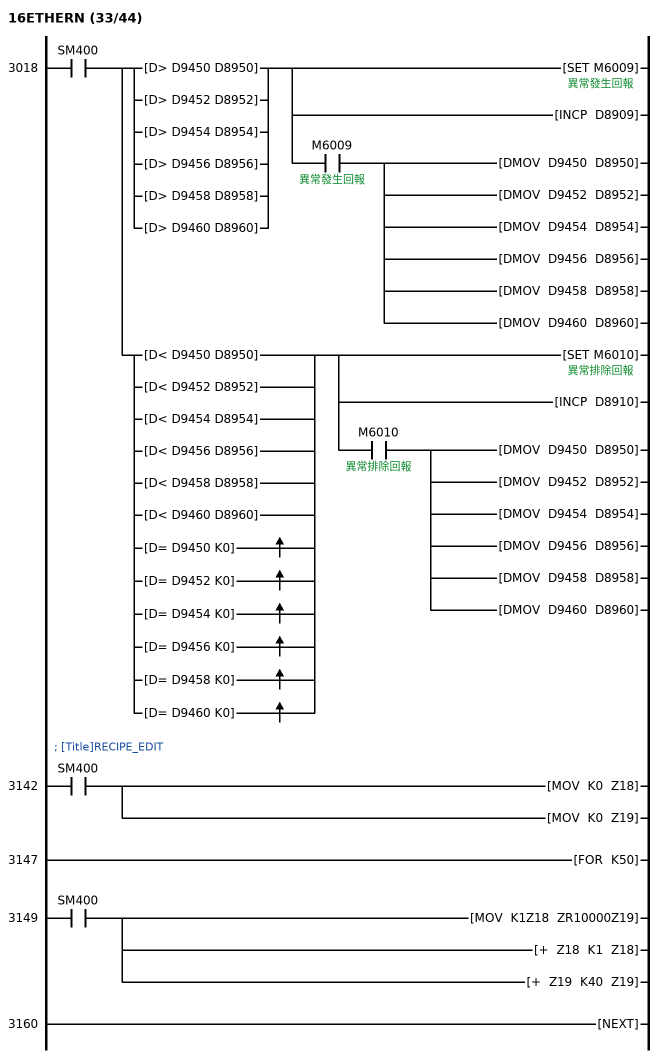
[picture p120: ladder of 16ETHERN, rungs at steps 3018 to 3160]
3018  LD      SM400
      MPS
      LDD>    D9450 D8950
      ORD>    D9452 D8952
      ORD>    D9454 D8954
      ORD>    D9456 D8956
      ORD>    D9458 D8958
      ORD>    D9460 D8960
      ANB
      SET     M6009  ; 異常發生回報
      INCP    D8909
      AND     M6009  ; 異常發生回報
      DMOV    D9450 D8950
      DMOV    D9452 D8952
      DMOV    D9454 D8954
      DMOV    D9456 D8956
      DMOV    D9458 D8958
      DMOV    D9460 D8960
      MPP
      LDD<    D9450 D8950
      ORD<    D9452 D8952
      ORD<    D9454 D8954
      ORD<    D9456 D8956
      ORD<    D9458 D8958
      ORD<    D9460 D8960
      LDD=    D9450 K0
      MEP
      ORB
      LDD=    D9452 K0
      MEP
      ORB
      LDD=    D9454 K0
      MEP
      ORB
      LDD=    D9456 K0
      MEP
      ORB
      LDD=    D9458 K0
      MEP
      ORB
      LDD=    D9460 K0
      MEP
      ORB
      ANB
      SET     M6010  ; 異常排除回報
      INCP    D8910
      AND     M6010  ; 異常排除回報
      DMOV    D9450 D8950
      DMOV    D9452 D8952
      DMOV    D9454 D8954
      DMOV    D9456 D8956
      DMOV    D9458 D8958
      DMOV    D9460 D8960
; [Title]RECIPE_EDIT
3142  LD      SM400
      MOV     K0 Z18
      MOV     K0 Z19
3147  FOR     K50
3149  LD      SM400
      MOV     K1Z18 ZR10000Z19
      +       Z18 K1 Z18
      +       Z19 K40 Z19
3160  NEXT
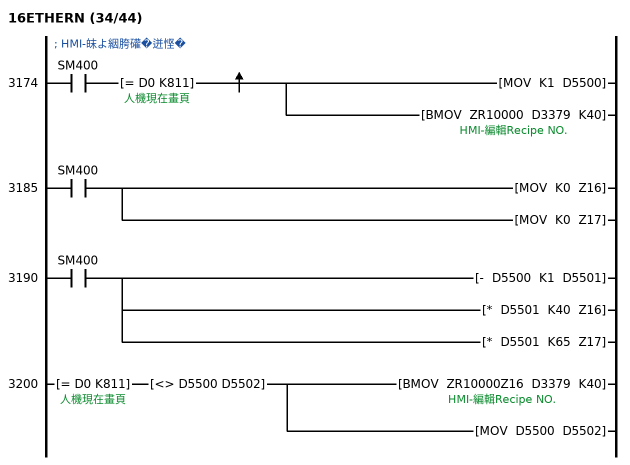
; HMI-配方編輯畫面顯示
3174  LD      SM400
      AND=    D0 K811  ; 人機現在畫頁
      MEP
      MOV     K1 D5500
      BMOV    ZR10000 D3379 K40  ; HMI-編輯Recipe NO.
3185  LD      SM400
      MOV     K0 Z16
      MOV     K0 Z17
3190  LD      SM400
      -       D5500 K1 D5501
      *       D5501 K40 Z16
      *       D5501 K65 Z17
3200  LD=     D0 K811  ; 人機現在畫頁
      AND<>   D5500 D5502
      BMOV    ZR10000Z16 D3379 K40
      MOV     D5500 D5502
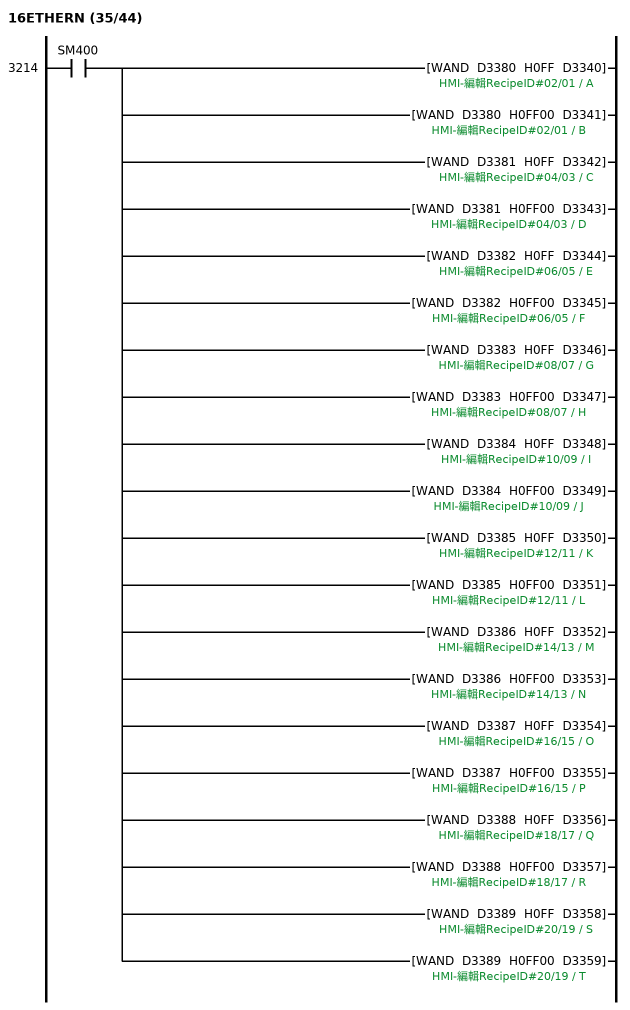
3214  LD      SM400
      WAND    D3380 H0FF D3340  ; HMI-編輯RecipeID#02/01 / A
      WAND    D3380 H0FF00 D3341  ; B
      WAND    D3381 H0FF D3342  ; HMI-編輯RecipeID#04/03 / C
      WAND    D3381 H0FF00 D3343  ; D
      WAND    D3382 H0FF D3344  ; HMI-編輯RecipeID#06/05 / E
      WAND    D3382 H0FF00 D3345  ; F
      WAND    D3383 H0FF D3346  ; HMI-編輯RecipeID#08/07 / G
      WAND    D3383 H0FF00 D3347  ; H
      WAND    D3384 H0FF D3348  ; HMI-編輯RecipeID#10/09 / I
      WAND    D3384 H0FF00 D3349  ; J
      WAND    D3385 H0FF D3350  ; HMI-編輯RecipeID#12/11 / K
      WAND    D3385 H0FF00 D3351  ; L
      WAND    D3386 H0FF D3352  ; HMI-編輯RecipeID#14/13 / M
      WAND    D3386 H0FF00 D3353  ; N
      WAND    D3387 H0FF D3354  ; HMI-編輯RecipeID#16/15 / O
      WAND    D3387 H0FF00 D3355  ; P
      WAND    D3388 H0FF D3356  ; HMI-編輯RecipeID#18/17 / Q
      WAND    D3388 H0FF00 D3357  ; R
      WAND    D3389 H0FF D3358  ; HMI-編輯RecipeID#20/19 / S
      WAND    D3389 H0FF00 D3359  ; T
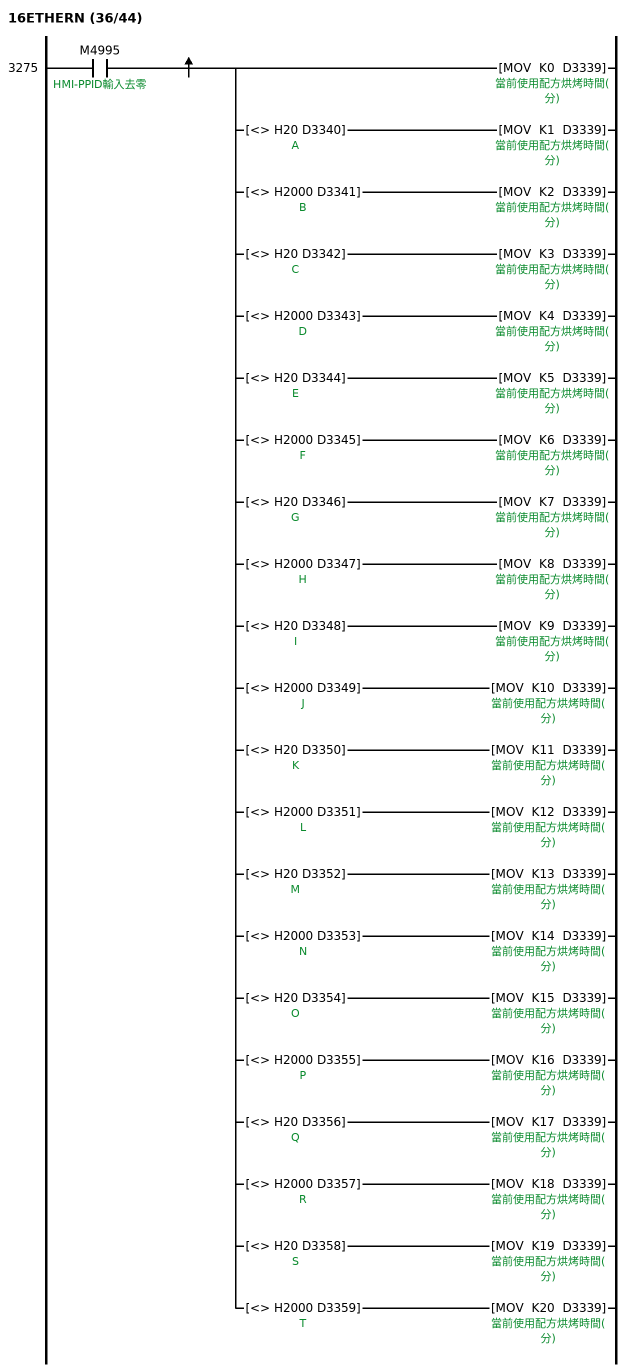
3275  LD      M4995  ; HMI-PPID輸入去零
      MEP
      MOV     K0 D3339  ; 當前使用配方烘烤時間(分)
      MPS
      AND<>   H20 D3340  ; A
      MOV     K1 D3339
      MRD
      AND<>   H2000 D3341  ; B
      MOV     K2 D3339
      MRD
      AND<>   H20 D3342  ; C
      MOV     K3 D3339
      MRD
      AND<>   H2000 D3343  ; D
      MOV     K4 D3339
      MRD
      AND<>   H20 D3344  ; E
      MOV     K5 D3339
      MRD
      AND<>   H2000 D3345  ; F
      MOV     K6 D3339
      MRD
      AND<>   H20 D3346  ; G
      MOV     K7 D3339
      MRD
      AND<>   H2000 D3347  ; H
      MOV     K8 D3339
      MRD
      AND<>   H20 D3348  ; I
      MOV     K9 D3339
      MRD
      AND<>   H2000 D3349  ; J
      MOV     K10 D3339
      MRD
      AND<>   H20 D3350  ; K
      MOV     K11 D3339
      MRD
      AND<>   H2000 D3351  ; L
      MOV     K12 D3339
      MRD
      AND<>   H20 D3352  ; M
      MOV     K13 D3339
      MRD
      AND<>   H2000 D3353  ; N
      MOV     K14 D3339
      MRD
      AND<>   H20 D3354  ; O
      MOV     K15 D3339
      MRD
      AND<>   H2000 D3355  ; P
      MOV     K16 D3339
      MRD
      AND<>   H20 D3356  ; Q
      MOV     K17 D3339
      MRD
      AND<>   H2000 D3357  ; R
      MOV     K18 D3339
      MRD
      AND<>   H20 D3358  ; S
      MOV     K19 D3339
      MPP
      AND<>   H2000 D3359  ; T
      MOV     K20 D3339
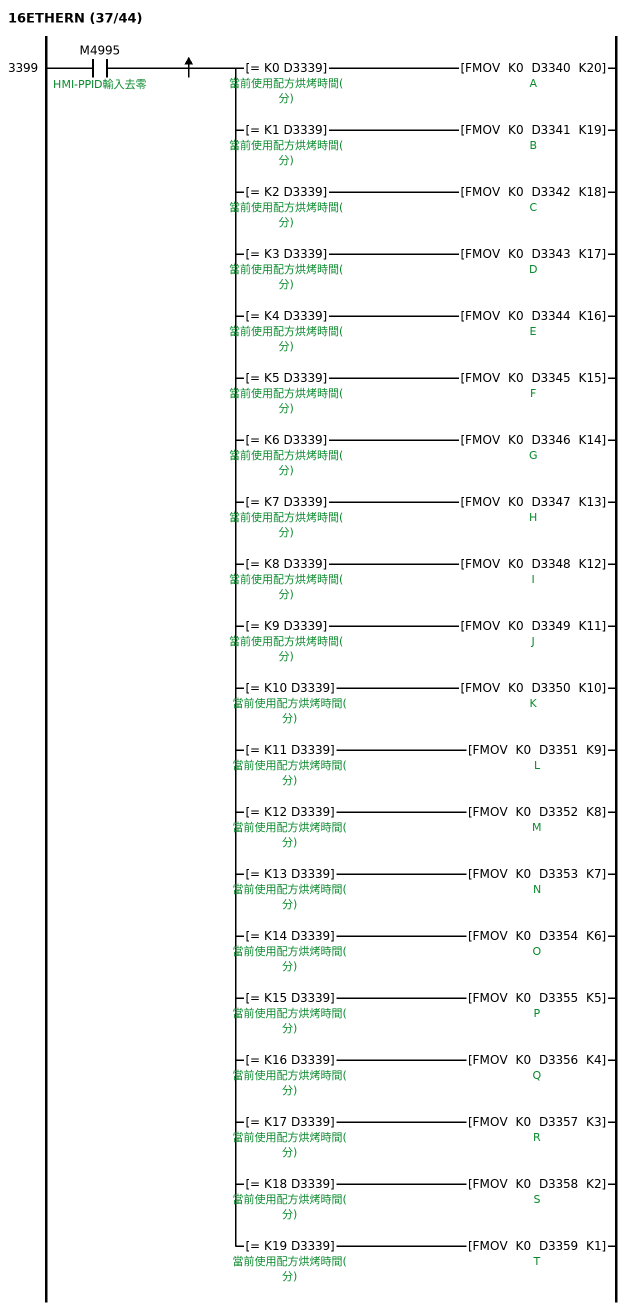
3399  LD      M4995  ; HMI-PPID輸入去零
      MEP
      MPS
      AND=    K0 D3339  ; 當前使用配方烘烤時間(分)
      FMOV    K0 D3340 K20
      MRD
      AND=    K1 D3339  ; 當前使用配方烘烤時間(分)
      FMOV    K0 D3341 K19
      MRD
      AND=    K2 D3339  ; 當前使用配方烘烤時間(分)
      FMOV    K0 D3342 K18
      MRD
      AND=    K3 D3339  ; 當前使用配方烘烤時間(分)
      FMOV    K0 D3343 K17
      MRD
      AND=    K4 D3339  ; 當前使用配方烘烤時間(分)
      FMOV    K0 D3344 K16
      MRD
      AND=    K5 D3339  ; 當前使用配方烘烤時間(分)
      FMOV    K0 D3345 K15
      MRD
      AND=    K6 D3339  ; 當前使用配方烘烤時間(分)
      FMOV    K0 D3346 K14
      MRD
      AND=    K7 D3339  ; 當前使用配方烘烤時間(分)
      FMOV    K0 D3347 K13
      MRD
      AND=    K8 D3339  ; 當前使用配方烘烤時間(分)
      FMOV    K0 D3348 K12
      MRD
      AND=    K9 D3339  ; 當前使用配方烘烤時間(分)
      FMOV    K0 D3349 K11
      MRD
      AND=    K10 D3339  ; 當前使用配方烘烤時間(分)
      FMOV    K0 D3350 K10
      MRD
      AND=    K11 D3339  ; 當前使用配方烘烤時間(分)
      FMOV    K0 D3351 K9
      MRD
      AND=    K12 D3339  ; 當前使用配方烘烤時間(分)
      FMOV    K0 D3352 K8
      MRD
      AND=    K13 D3339  ; 當前使用配方烘烤時間(分)
      FMOV    K0 D3353 K7
      MRD
      AND=    K14 D3339  ; 當前使用配方烘烤時間(分)
      FMOV    K0 D3354 K6
      MRD
      AND=    K15 D3339  ; 當前使用配方烘烤時間(分)
      FMOV    K0 D3355 K5
      MRD
      AND=    K16 D3339  ; 當前使用配方烘烤時間(分)
      FMOV    K0 D3356 K4
      MRD
      AND=    K17 D3339  ; 當前使用配方烘烤時間(分)
      FMOV    K0 D3357 K3
      MRD
      AND=    K18 D3339  ; 當前使用配方烘烤時間(分)
      FMOV    K0 D3358 K2
      MPP
      AND=    K19 D3339  ; 當前使用配方烘烤時間(分)
      FMOV    K0 D3359 K1
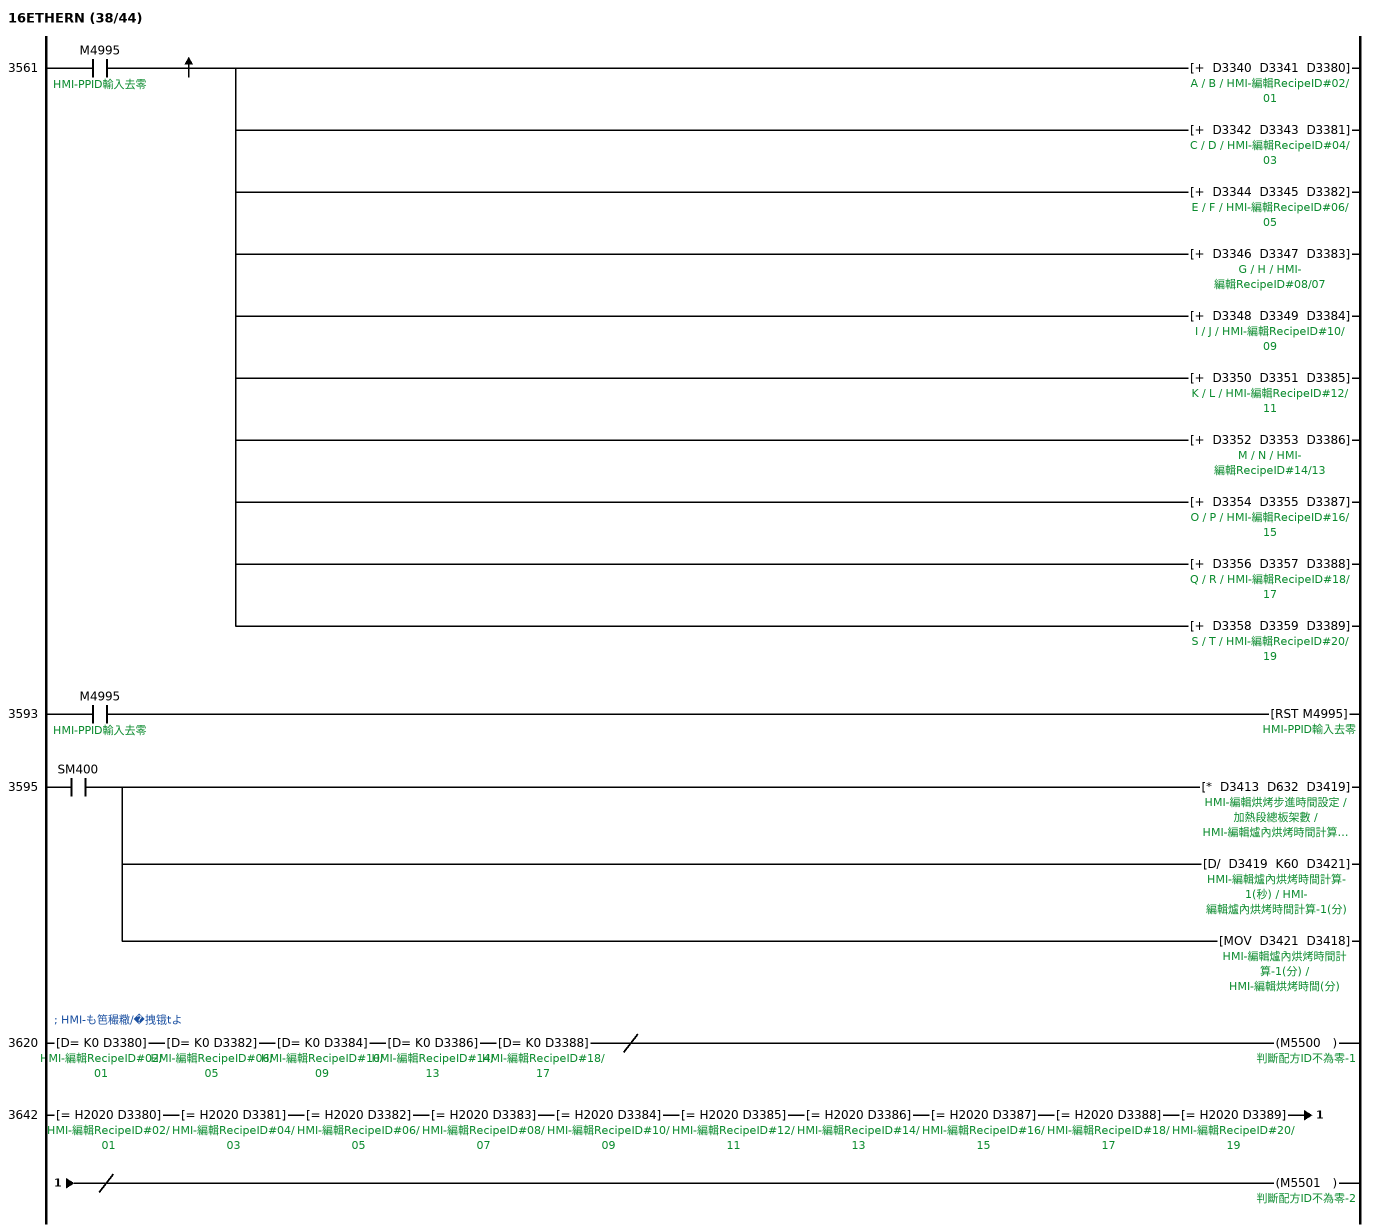
3561  LD      M4995  ; HMI-PPID輸入去零
      MEP
      +       D3340 D3341 D3380
      +       D3342 D3343 D3381
      +       D3344 D3345 D3382
      +       D3346 D3347 D3383
      +       D3348 D3349 D3384
      +       D3350 D3351 D3385
      +       D3352 D3353 D3386
      +       D3354 D3355 D3387
      +       D3356 D3357 D3388
      +       D3358 D3359 D3389
3593  LD      M4995  ; HMI-PPID輸入去零
      RST     M4995  ; HMI-PPID輸入去零
3595  LD      SM400
      *       D3413 D632 D3419  ; HMI-編輯烘烤步進時間設定 / 加熱段總板架數 / HMI-編輯爐內烘烤時間計算-1(秒)
      D/      D3419 K60 D3421  ; HMI-編輯爐內烘烤時間計算-1(分)
      MOV     D3421 D3418  ; HMI-編輯烘烤時間(分)
; HMI-手動新增/修改配方
3620  LDD=    K0 D3380  ; HMI-編輯RecipeID#02/01
      ANDD=   K0 D3382  ; HMI-編輯RecipeID#06/05
      ANDD=   K0 D3384  ; HMI-編輯RecipeID#10/09
      ANDD=   K0 D3386  ; HMI-編輯RecipeID#14/13
      ANDD=   K0 D3388  ; HMI-編輯RecipeID#18/17
      INV
      OUT     M5500  ; 判斷配方ID不為零-1
3642  LD=     H2020 D3380  ; HMI-編輯RecipeID#02/01
      AND=    H2020 D3381  ; HMI-編輯RecipeID#04/03
      AND=    H2020 D3382  ; HMI-編輯RecipeID#06/05
      AND=    H2020 D3383  ; HMI-編輯RecipeID#08/07
      AND=    H2020 D3384  ; HMI-編輯RecipeID#10/09
      AND=    H2020 D3385  ; HMI-編輯RecipeID#12/11
      AND=    H2020 D3386  ; HMI-編輯RecipeID#14/13
      AND=    H2020 D3387  ; HMI-編輯RecipeID#16/15
      AND=    H2020 D3388  ; HMI-編輯RecipeID#18/17
      AND=    H2020 D3389  ; HMI-編輯RecipeID#20/19
      INV
      OUT     M5501  ; 判斷配方ID不為零-2
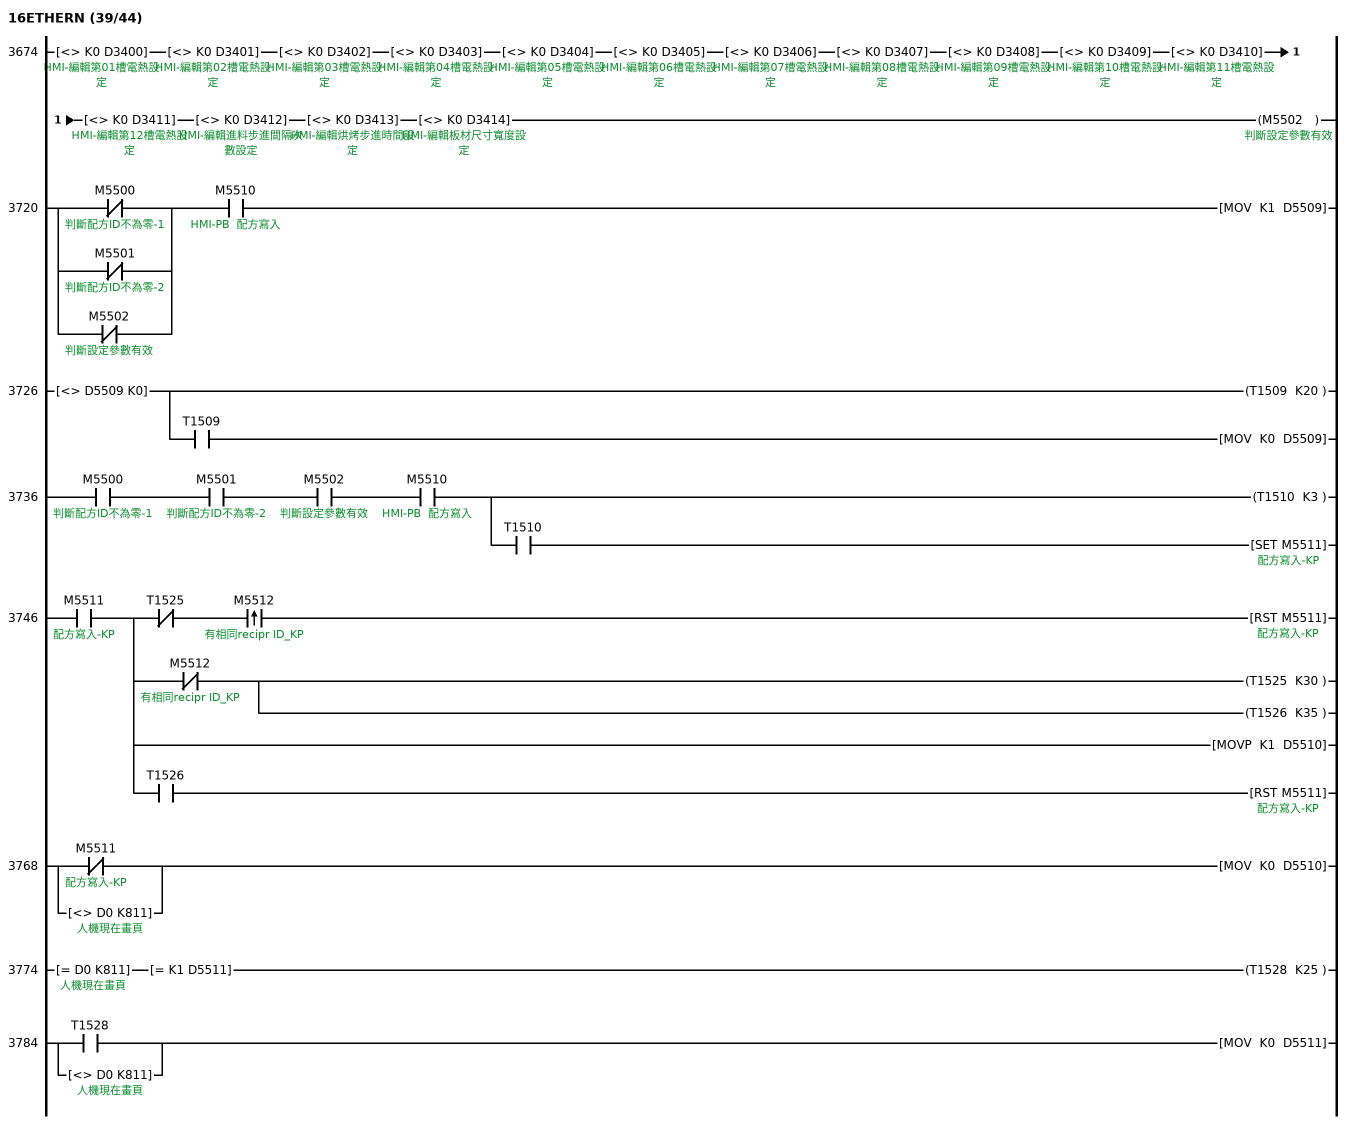
3674  LD<>    K0 D3400  ; HMI-編輯第01槽電熱設定
      AND<>   K0 D3401  ; HMI-編輯第02槽電熱設定
      AND<>   K0 D3402  ; HMI-編輯第03槽電熱設定
      AND<>   K0 D3403  ; HMI-編輯第04槽電熱設定
      AND<>   K0 D3404  ; HMI-編輯第05槽電熱設定
      AND<>   K0 D3405  ; HMI-編輯第06槽電熱設定
      AND<>   K0 D3406  ; HMI-編輯第07槽電熱設定
      AND<>   K0 D3407  ; HMI-編輯第08槽電熱設定
      AND<>   K0 D3408  ; HMI-編輯第09槽電熱設定
      AND<>   K0 D3409  ; HMI-編輯第10槽電熱設定
      AND<>   K0 D3410  ; HMI-編輯第11槽電熱設定
      AND<>   K0 D3411  ; HMI-編輯第12槽電熱設定
      AND<>   K0 D3412  ; HMI-編輯進料步進間隔次數設定
      AND<>   K0 D3413  ; HMI-編輯烘烤步進時間設定
      AND<>   K0 D3414  ; HMI-編輯板材尺寸寬度設定
      OUT     M5502  ; 判斷設定參數有效
3720  LDI     M5500  ; 判斷配方ID不為零-1
      ORI     M5501  ; 判斷配方ID不為零-2
      ORI     M5502  ; 判斷設定參數有效
      AND     M5510  ; HMI-PB  配方寫入
      MOV     K1 D5509
3726  LD<>    D5509 K0
      OUT     T1509 K20
      AND     T1509
      MOV     K0 D5509
3736  LD      M5500  ; 判斷配方ID不為零-1
      AND     M5501  ; 判斷配方ID不為零-2
      AND     M5502  ; 判斷設定參數有效
      AND     M5510  ; HMI-PB  配方寫入
      OUT     T1510 K3
      AND     T1510
      SET     M5511  ; 配方寫入-KP
3746  LD      M5511  ; 配方寫入-KP
      MPS
      ANI     T1525
      ANDP    M5512  ; 有相同recipr ID_KP
      RST     M5511  ; 配方寫入-KP
      MRD
      ANI     M5512  ; 有相同recipr ID_KP
      OUT     T1525 K30
      OUT     T1526 K35
      MPP
      MOVP    K1 D5510
      AND     T1526
      RST     M5511  ; 配方寫入-KP
3768  LDI     M5511  ; 配方寫入-KP
      OR<>    D0 K811  ; 人機現在畫頁
      MOV     K0 D5510
3774  LD=     D0 K811  ; 人機現在畫頁
      AND=    K1 D5511
      OUT     T1528 K25
3784  LD      T1528
      OR<>    D0 K811  ; 人機現在畫頁
      MOV     K0 D5511
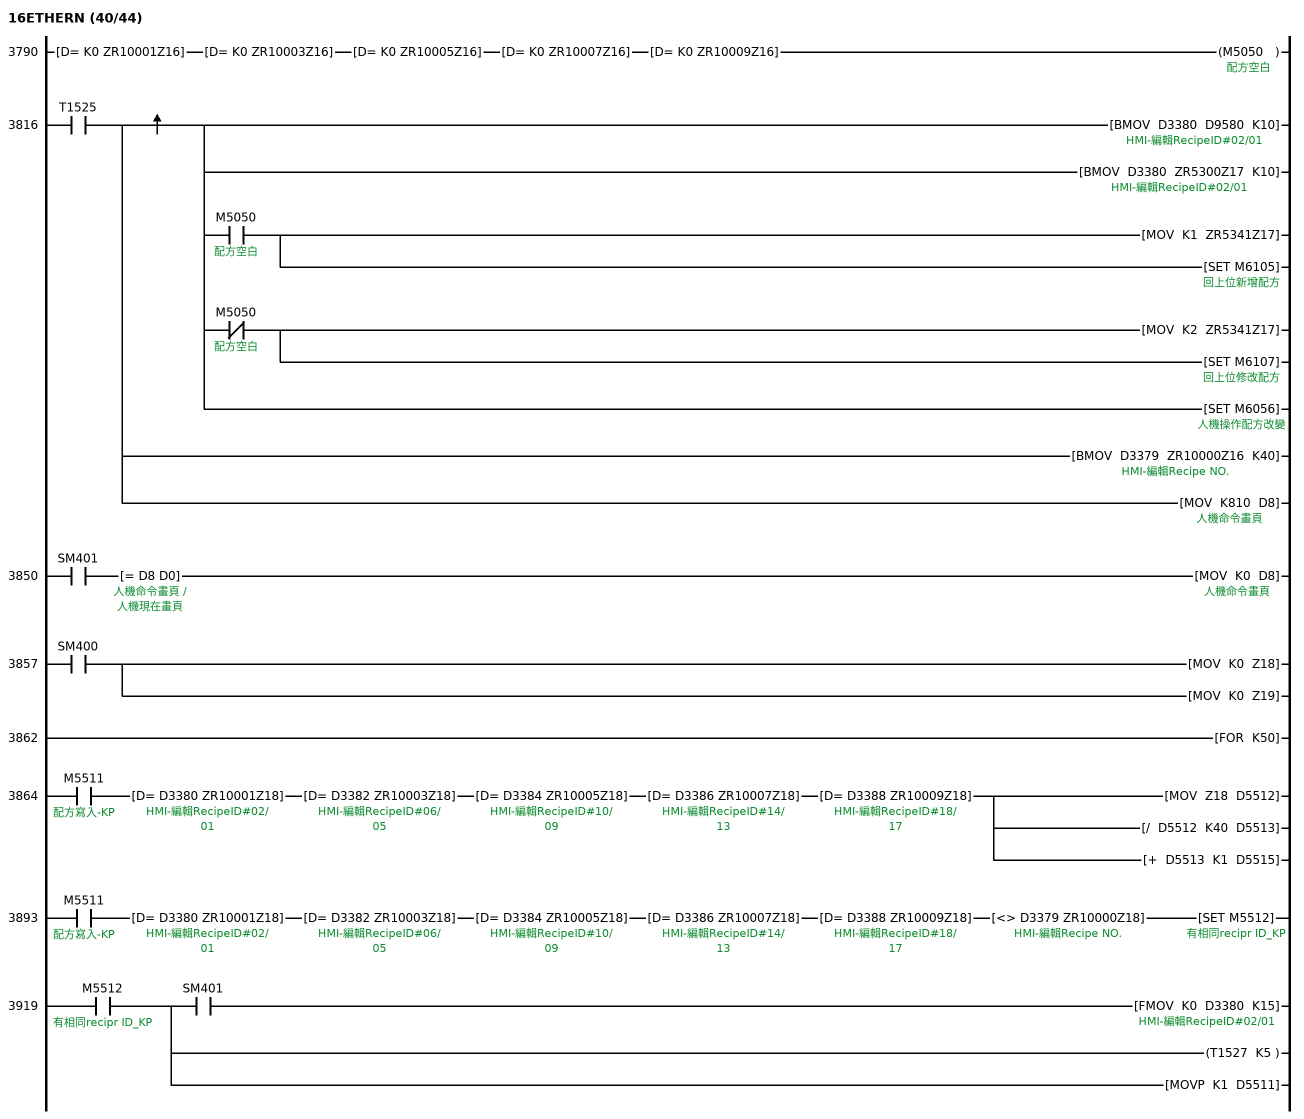
3790  LDD=    K0 ZR10001Z16
      ANDD=   K0 ZR10003Z16
      ANDD=   K0 ZR10005Z16
      ANDD=   K0 ZR10007Z16
      ANDD=   K0 ZR10009Z16
      OUT     M5050  ; 配方空白
3816  LD      T1525
      MPS
      MEP
      BMOV    D3380 D9580 K10
      BMOV    D3380 ZR5300Z17 K10
      MPS
      AND     M5050  ; 配方空白
      MOV     K1 ZR5341Z17
      SET     M6105  ; 回上位新增配方
      MRD
      ANI     M5050  ; 配方空白
      MOV     K2 ZR5341Z17
      SET     M6107  ; 回上位修改配方
      MPP
      SET     M6056  ; 人機操作配方改變
      MPP
      BMOV    D3379 ZR10000Z16 K40
      MOV     K810 D8
3850  LD      SM401
      AND=    D8 D0  ; 人機命令畫頁 / 人機現在畫頁
      MOV     K0 D8
3857  LD      SM400
      MOV     K0 Z18
      MOV     K0 Z19
3862  FOR     K50
3864  LD      M5511  ; 配方寫入-KP
      ANDD=   D3380 ZR10001Z18  ; HMI-編輯RecipeID#02/01
      ANDD=   D3382 ZR10003Z18  ; HMI-編輯RecipeID#06/05
      ANDD=   D3384 ZR10005Z18  ; HMI-編輯RecipeID#10/09
      ANDD=   D3386 ZR10007Z18  ; HMI-編輯RecipeID#14/13
      ANDD=   D3388 ZR10009Z18  ; HMI-編輯RecipeID#18/17
      MOV     Z18 D5512
      /       D5512 K40 D5513
      +       D5513 K1 D5515
3893  LD      M5511  ; 配方寫入-KP
      ANDD=   D3380 ZR10001Z18  ; HMI-編輯RecipeID#02/01
      ANDD=   D3382 ZR10003Z18  ; HMI-編輯RecipeID#06/05
      ANDD=   D3384 ZR10005Z18  ; HMI-編輯RecipeID#10/09
      ANDD=   D3386 ZR10007Z18  ; HMI-編輯RecipeID#14/13
      ANDD=   D3388 ZR10009Z18  ; HMI-編輯RecipeID#18/17
      AND<>   D3379 ZR10000Z18  ; HMI-編輯Recipe NO.
      SET     M5512  ; 有相同recipr ID_KP
3919  LD      M5512  ; 有相同recipr ID_KP
      MPS
      AND     SM401
      FMOV    K0 D3380 K15
      MPP
      OUT     T1527 K5
      MOVP    K1 D5511
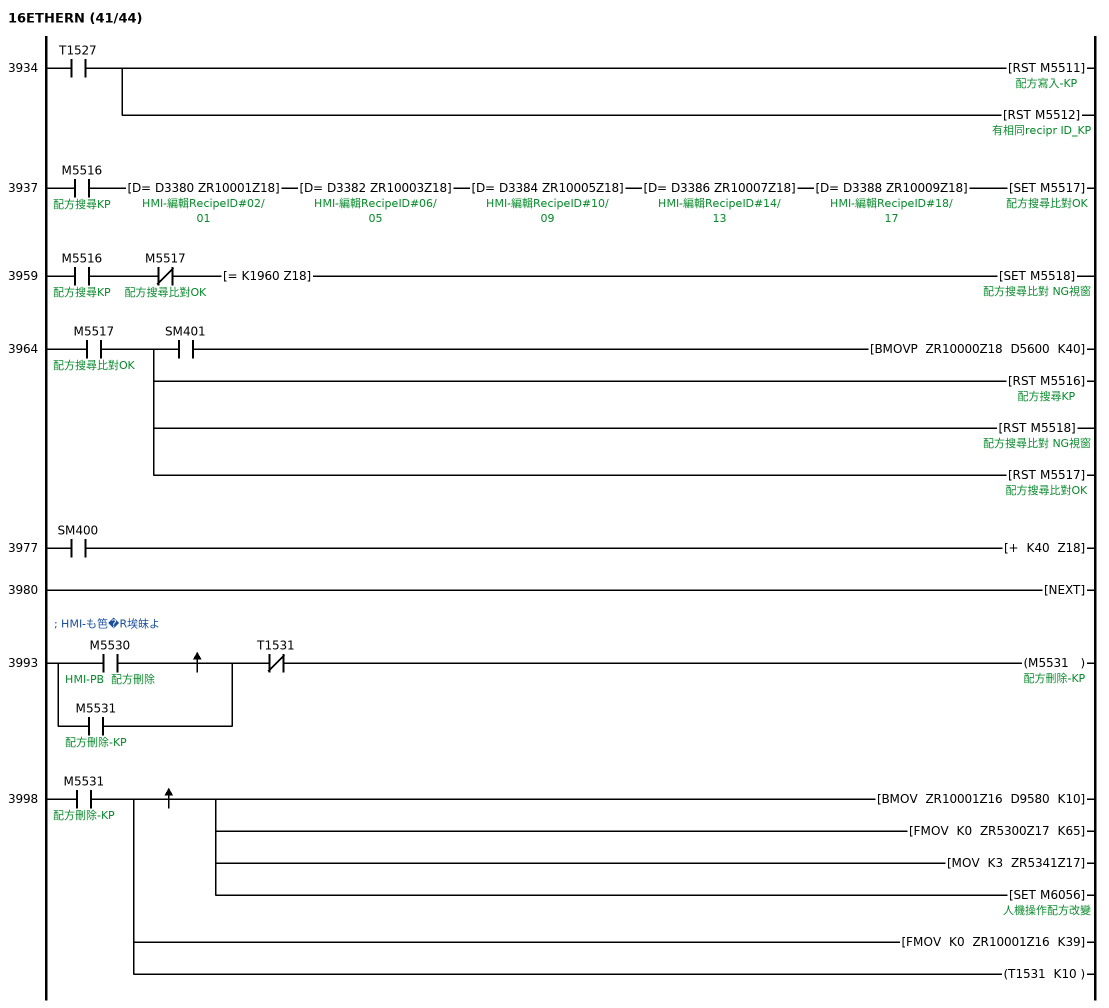
3934  LD      T1527
      RST     M5511  ; 配方寫入-KP
      RST     M5512  ; 有相同recipr ID_KP
3937  LD      M5516  ; 配方搜尋KP
      ANDD=   D3380 ZR10001Z18  ; HMI-編輯RecipeID#02/01
      ANDD=   D3382 ZR10003Z18  ; HMI-編輯RecipeID#06/05
      ANDD=   D3384 ZR10005Z18  ; HMI-編輯RecipeID#10/09
      ANDD=   D3386 ZR10007Z18  ; HMI-編輯RecipeID#14/13
      ANDD=   D3388 ZR10009Z18  ; HMI-編輯RecipeID#18/17
      SET     M5517  ; 配方搜尋比對OK
3959  LD      M5516  ; 配方搜尋KP
      ANI     M5517  ; 配方搜尋比對OK
      AND=    K1960 Z18
      SET     M5518  ; 配方搜尋比對 NG視窗
3964  LD      M5517  ; 配方搜尋比對OK
      MPS
      AND     SM401
      BMOVP   ZR10000Z18 D5600 K40
      MPP
      RST     M5516  ; 配方搜尋KP
      RST     M5518  ; 配方搜尋比對 NG視窗
      RST     M5517  ; 配方搜尋比對OK
3977  LD      SM400
      +       K40 Z18
3980  NEXT
; HMI-手動刪除配方
3993  LD      M5530  ; HMI-PB  配方刪除
      MEP
      OR      M5531  ; 配方刪除-KP
      ANI     T1531
      OUT     M5531  ; 配方刪除-KP
3998  LD      M5531  ; 配方刪除-KP
      MPS
      MEP
      BMOV    ZR10001Z16 D9580 K10
      FMOV    K0 ZR5300Z17 K65
      MOV     K3 ZR5341Z17
      SET     M6056  ; 人機操作配方改變
      MPP
      FMOV    K0 ZR10001Z16 K39
      OUT     T1531 K10
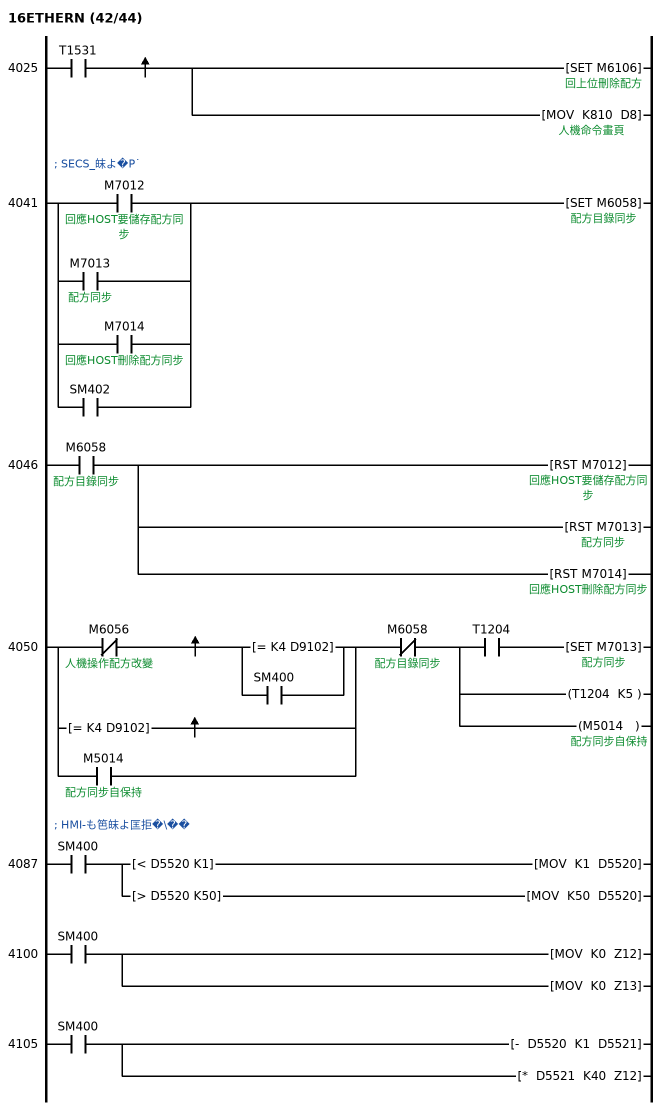
4025  LD      T1531
      MEP
      SET     M6106  ; 回上位刪除配方
      MOV     K810 D8
; SECS_配方同步
4041  LD      M7012  ; 回應HOST要儲存配方同步
      OR      M7013  ; 配方同步
      OR      M7014  ; 回應HOST刪除配方同步
      OR      SM402
      SET     M6058  ; 配方目錄同步
4046  LD      M6058  ; 配方目錄同步
      RST     M7012  ; 回應HOST要儲存配方同步
      RST     M7013  ; 配方同步
      RST     M7014  ; 回應HOST刪除配方同步
4050  LDI     M6056  ; 人機操作配方改變
      MEP
      LD=     K4 D9102
      OR      SM400
      ANB
      LD=     K4 D9102
      MEP
      ORB
      OR      M5014  ; 配方同步自保持
      ANI     M6058  ; 配方目錄同步
      MPS
      AND     T1204
      SET     M7013  ; 配方同步
      MPP
      OUT     T1204 K5
      OUT     M5014  ; 配方同步自保持
; HMI-手動配方選擇功能
4087  LD      SM400
      MPS
      AND<    D5520 K1
      MOV     K1 D5520
      MPP
      AND>    D5520 K50
      MOV     K50 D5520
4100  LD      SM400
      MOV     K0 Z12
      MOV     K0 Z13
4105  LD      SM400
      -       D5520 K1 D5521
      *       D5521 K40 Z12
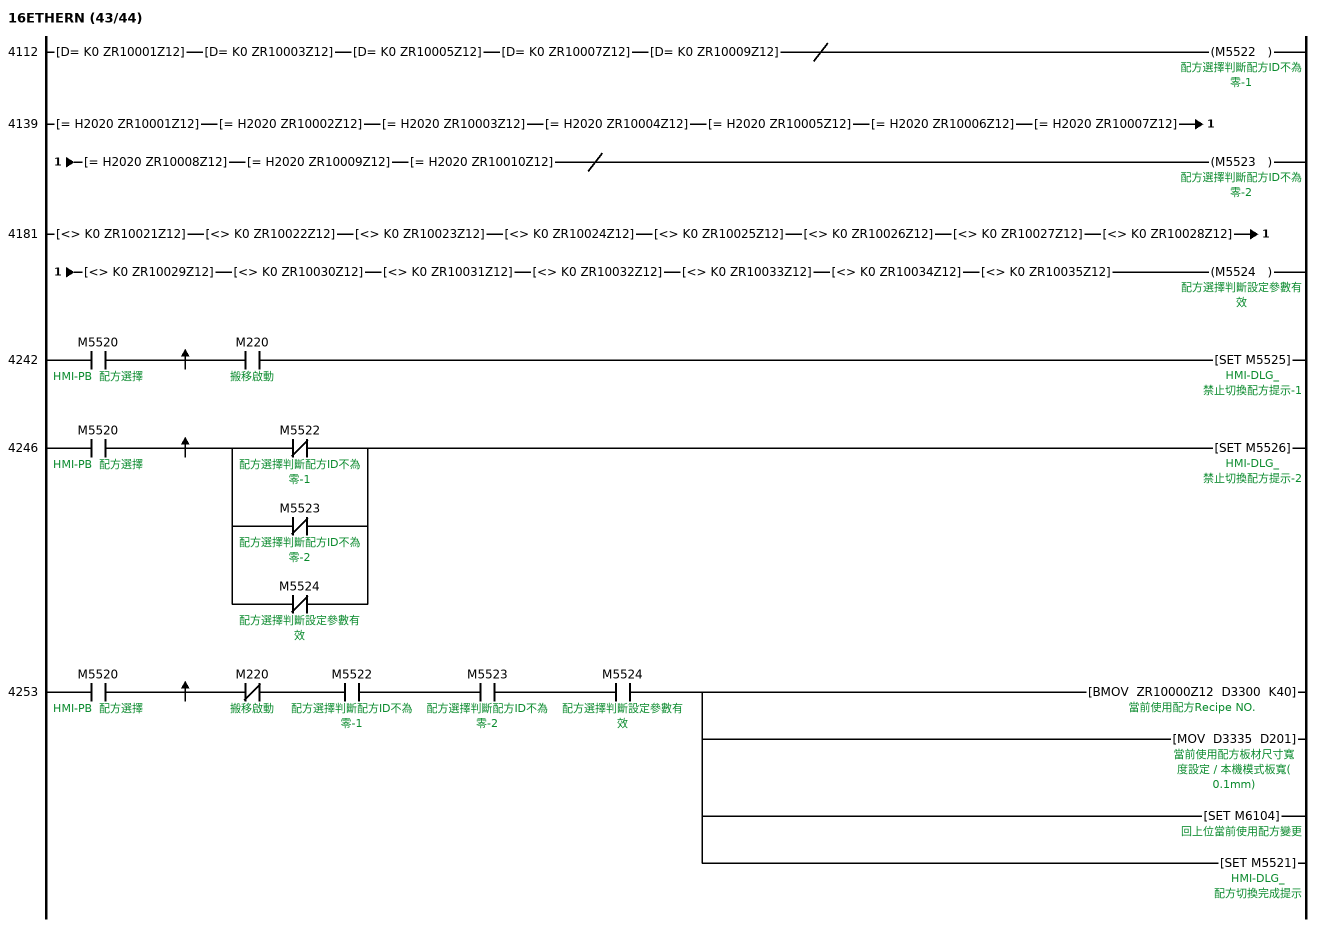
4112  LDD=    K0 ZR10001Z12
      ANDD=   K0 ZR10003Z12
      ANDD=   K0 ZR10005Z12
      ANDD=   K0 ZR10007Z12
      ANDD=   K0 ZR10009Z12
      INV
      OUT     M5522  ; 配方選擇判斷配方ID不為零-1
4139  LD=     H2020 ZR10001Z12
      AND=    H2020 ZR10002Z12
      AND=    H2020 ZR10003Z12
      AND=    H2020 ZR10004Z12
      AND=    H2020 ZR10005Z12
      AND=    H2020 ZR10006Z12
      AND=    H2020 ZR10007Z12
      AND=    H2020 ZR10008Z12
      AND=    H2020 ZR10009Z12
      AND=    H2020 ZR10010Z12
      INV
      OUT     M5523  ; 配方選擇判斷配方ID不為零-2
4181  LD<>    K0 ZR10021Z12
      AND<>   K0 ZR10022Z12
      AND<>   K0 ZR10023Z12
      AND<>   K0 ZR10024Z12
      AND<>   K0 ZR10025Z12
      AND<>   K0 ZR10026Z12
      AND<>   K0 ZR10027Z12
      AND<>   K0 ZR10028Z12
      AND<>   K0 ZR10029Z12
      AND<>   K0 ZR10030Z12
      AND<>   K0 ZR10031Z12
      AND<>   K0 ZR10032Z12
      AND<>   K0 ZR10033Z12
      AND<>   K0 ZR10034Z12
      AND<>   K0 ZR10035Z12
      OUT     M5524  ; 配方選擇判斷設定參數有效
4242  LD      M5520  ; HMI-PB  配方選擇
      MEP
      AND     M220  ; 搬移啟動
      SET     M5525  ; HMI-DLG_禁止切換配方提示-1
4246  LD      M5520  ; HMI-PB  配方選擇
      MEP
      LDI     M5522  ; 配方選擇判斷配方ID不為零-1
      ORI     M5523  ; 配方選擇判斷配方ID不為零-2
      ORI     M5524  ; 配方選擇判斷設定參數有效
      ANB
      SET     M5526  ; HMI-DLG_禁止切換配方提示-2
4253  LD      M5520  ; HMI-PB  配方選擇
      MEP
      ANI     M220  ; 搬移啟動
      AND     M5522  ; 配方選擇判斷配方ID不為零-1
      AND     M5523  ; 配方選擇判斷配方ID不為零-2
      AND     M5524  ; 配方選擇判斷設定參數有效
      BMOV    ZR10000Z12 D3300 K40
      MOV     D3335 D201
      SET     M6104  ; 回上位當前使用配方變更
      SET     M5521  ; HMI-DLG_配方切換完成提示
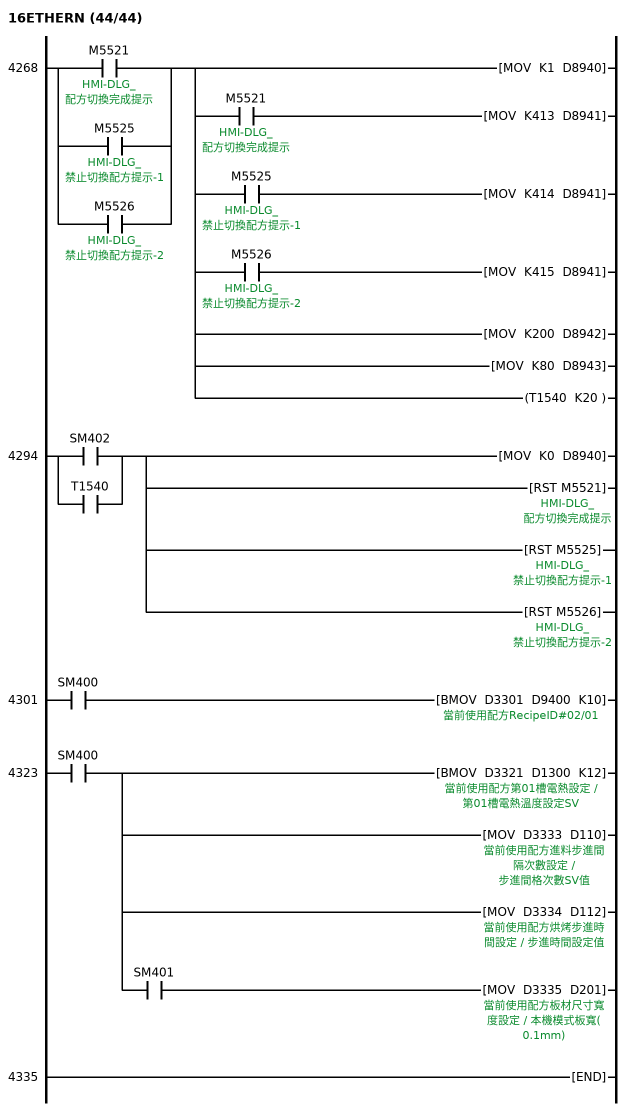
4268  LD      M5521  ; HMI-DLG_配方切換完成提示
      OR      M5525  ; HMI-DLG_禁止切換配方提示-1
      OR      M5526  ; HMI-DLG_禁止切換配方提示-2
      MOV     K1 D8940
      MPS
      AND     M5521  ; HMI-DLG_配方切換完成提示
      MOV     K413 D8941
      MRD
      AND     M5525  ; HMI-DLG_禁止切換配方提示-1
      MOV     K414 D8941
      MRD
      AND     M5526  ; HMI-DLG_禁止切換配方提示-2
      MOV     K415 D8941
      MPP
      MOV     K200 D8942
      MOV     K80 D8943
      OUT     T1540 K20
4294  LD      SM402
      OR      T1540
      MOV     K0 D8940
      RST     M5521  ; HMI-DLG_配方切換完成提示
      RST     M5525  ; HMI-DLG_禁止切換配方提示-1
      RST     M5526  ; HMI-DLG_禁止切換配方提示-2
4301  LD      SM400
      BMOV    D3301 D9400 K10  ; 當前使用配方RecipeID#02/01
        [note] D9400_上報SECS目前使用PPID名稱
4323  LD      SM400
      BMOV    D3321 D1300 K12  ; 當前使用配方第01槽電熱設定
      MOV     D3333 D110  ; 當前使用配方進料步進間隔次數設定
      MOV     D3334 D112  ; 當前使用配方烘烤步進時間設定
      AND     SM401
      MOV     D3335 D201
4335  END
END_PROGRAM

PROGRAM 17GBF-20
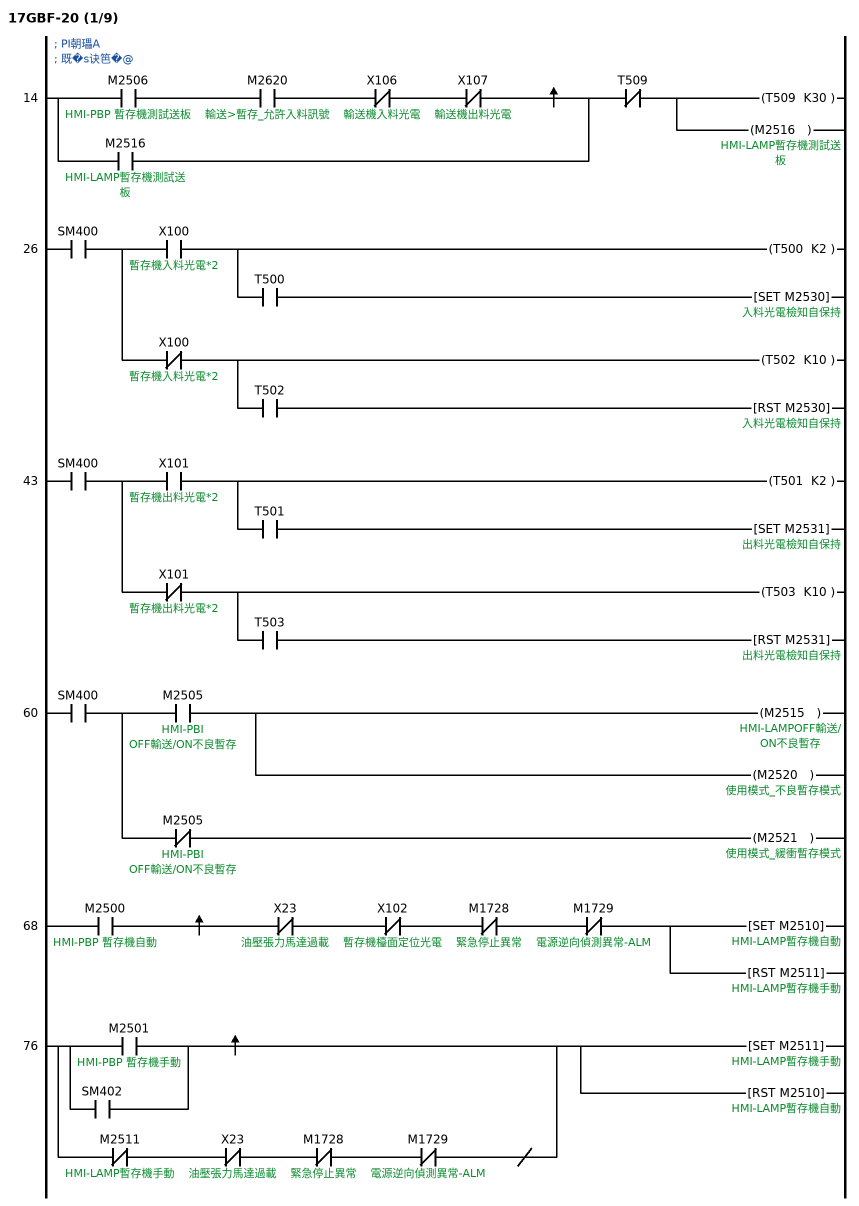
; PI朝瓃Α
; 暫存機動作
14    LD      M2506  ; HMI-PBP 暫存機測試送板
      AND     M2620  ; 輸送>暫存_允許入料訊號
      ANI     X106  ; 輸送機入料光電
      ANI     X107  ; 輸送機出料光電
      MEP
      OR      M2516  ; HMI-LAMP暫存機測試送板
      ANI     T509
      OUT     T509 K30
      OUT     M2516  ; HMI-LAMP暫存機測試送板
26    LD      SM400
      MPS
      AND     X100  ; 暫存機入料光電*2
      OUT     T500 K2
      AND     T500
      SET     M2530  ; 入料光電檢知自保持
      MPP
      ANI     X100  ; 暫存機入料光電*2
      OUT     T502 K10
      AND     T502
      RST     M2530  ; 入料光電檢知自保持
43    LD      SM400
      MPS
      AND     X101  ; 暫存機出料光電*2
      OUT     T501 K2
      AND     T501
      SET     M2531  ; 出料光電檢知自保持
      MPP
      ANI     X101  ; 暫存機出料光電*2
      OUT     T503 K10
      AND     T503
      RST     M2531  ; 出料光電檢知自保持
60    LD      SM400
      MPS
      AND     M2505  ; HMI-PBI OFF輸送/ON不良暫存
      OUT     M2515  ; HMI-LAMPOFF輸送/ON不良暫存
      OUT     M2520  ; 使用模式_不良暫存模式
      MPP
      ANI     M2505  ; HMI-PBI OFF輸送/ON不良暫存
      OUT     M2521  ; 使用模式_緩衝暫存模式
68    LD      M2500  ; HMI-PBP 暫存機自動
      MEP
      ANI     X23  ; 油壓張力馬達過載
      ANI     X102  ; 暫存機檯面定位光電
      ANI     M1728  ; 緊急停止異常
      ANI     M1729  ; 電源逆向偵測異常-ALM
      SET     M2510  ; HMI-LAMP暫存機自動
      RST     M2511  ; HMI-LAMP暫存機手動
76    LD      M2501  ; HMI-PBP 暫存機手動
      OR      SM402
      MEP
      LDI     M2511  ; HMI-LAMP暫存機手動
      ANI     X23  ; 油壓張力馬達過載
      ANI     M1728  ; 緊急停止異常
      ANI     M1729  ; 電源逆向偵測異常-ALM
      INV
      ORB
      SET     M2511  ; HMI-LAMP暫存機手動
      RST     M2510  ; HMI-LAMP暫存機自動
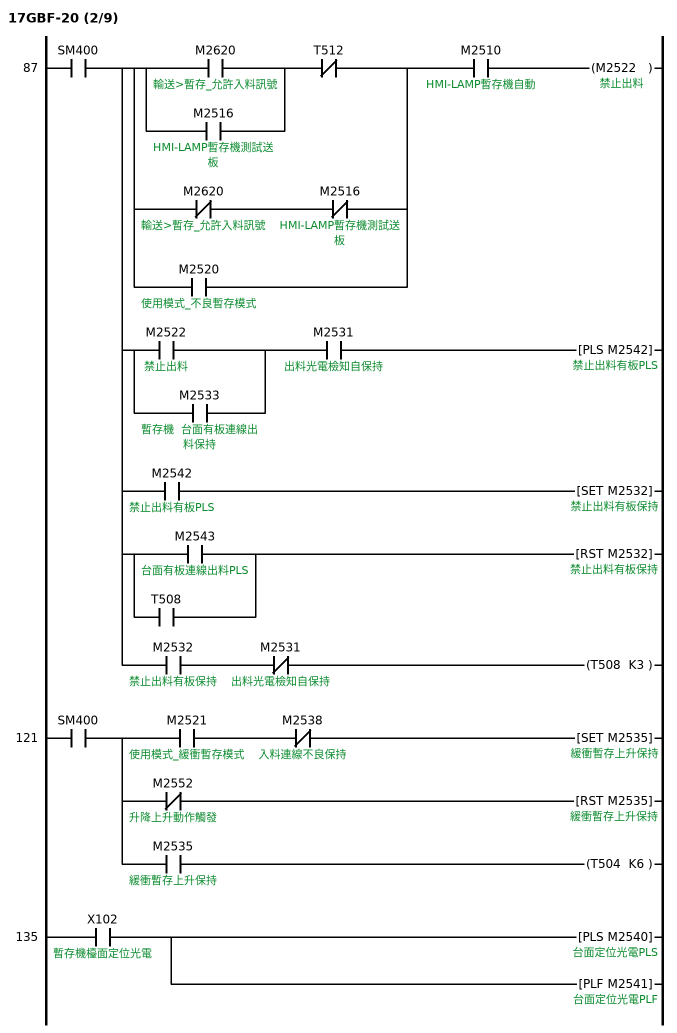
87    LD      SM400
      MPS
      LD      M2620  ; 輸送>暫存_允許入料訊號
      OR      M2516  ; HMI-LAMP暫存機測試送板
      ANI     T512
      LDI     M2620  ; 輸送>暫存_允許入料訊號
      ANI     M2516  ; HMI-LAMP暫存機測試送板
      ORB
      OR      M2520  ; 使用模式_不良暫存模式
      ANB
      AND     M2510  ; HMI-LAMP暫存機自動
      OUT     M2522  ; 禁止出料
      MRD
      LD      M2522  ; 禁止出料
      OR      M2533  ; 暫存機  台面有板連線出料保持
      ANB
      AND     M2531  ; 出料光電檢知自保持
      PLS     M2542  ; 禁止出料有板PLS
      MRD
      AND     M2542  ; 禁止出料有板PLS
      SET     M2532  ; 禁止出料有板保持
      MRD
      LD      M2543  ; 台面有板連線出料PLS
      OR      T508
      ANB
      RST     M2532  ; 禁止出料有板保持
      MPP
      AND     M2532  ; 禁止出料有板保持
      ANI     M2531  ; 出料光電檢知自保持
      OUT     T508 K3
121   LD      SM400
      MPS
      AND     M2521  ; 使用模式_緩衝暫存模式
      ANI     M2538  ; 入料連線不良保持
      SET     M2535  ; 緩衝暫存上升保持
      MRD
      ANI     M2552  ; 升降上升動作觸發
      RST     M2535  ; 緩衝暫存上升保持
      MPP
      AND     M2535  ; 緩衝暫存上升保持
      OUT     T504 K6
135   LD      X102  ; 暫存機檯面定位光電
      PLS     M2540  ; 台面定位光電PLS
      PLF     M2541  ; 台面定位光電PLF
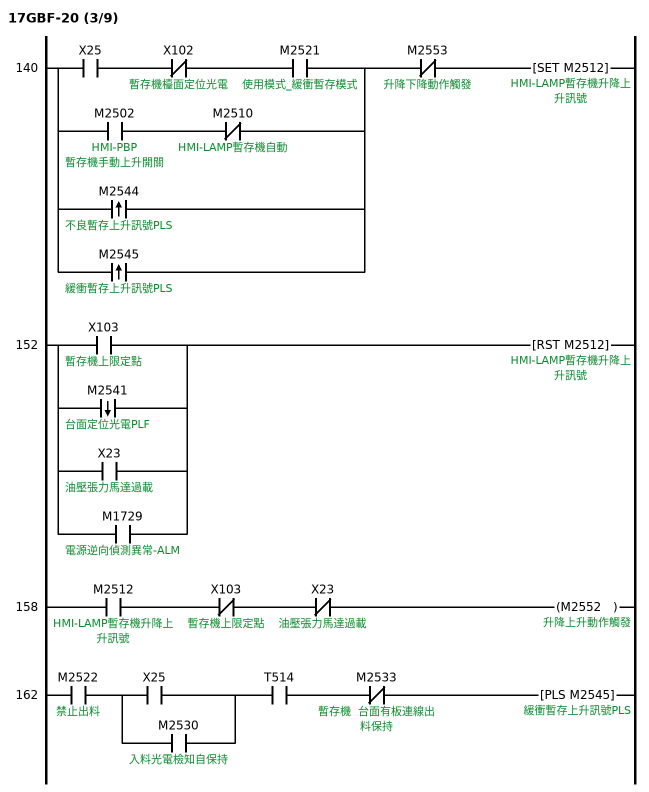
140   LD      X25
      ANI     X102  ; 暫存機檯面定位光電
      AND     M2521  ; 使用模式_緩衝暫存模式
      LD      M2502  ; HMI-PBP 暫存機手動上升開關
      ANI     M2510  ; HMI-LAMP暫存機自動
      ORB
      ORP     M2544  ; 不良暫存上升訊號PLS
      ORP     M2545  ; 緩衝暫存上升訊號PLS
      ANI     M2553  ; 升降下降動作觸發
      SET     M2512  ; HMI-LAMP暫存機升降上升訊號
152   LD      X103  ; 暫存機上限定點
      ORF     M2541  ; 台面定位光電PLF
      OR      X23  ; 油壓張力馬達過載
      OR      M1729  ; 電源逆向偵測異常-ALM
      RST     M2512  ; HMI-LAMP暫存機升降上升訊號
158   LD      M2512  ; HMI-LAMP暫存機升降上升訊號
      ANI     X103  ; 暫存機上限定點
      ANI     X23  ; 油壓張力馬達過載
      OUT     M2552  ; 升降上升動作觸發
162   LD      M2522  ; 禁止出料
      LD      X25
      OR      M2530  ; 入料光電檢知自保持
      ANB
      AND     T514
      ANI     M2533  ; 暫存機  台面有板連線出料保持
      PLS     M2545  ; 緩衝暫存上升訊號PLS
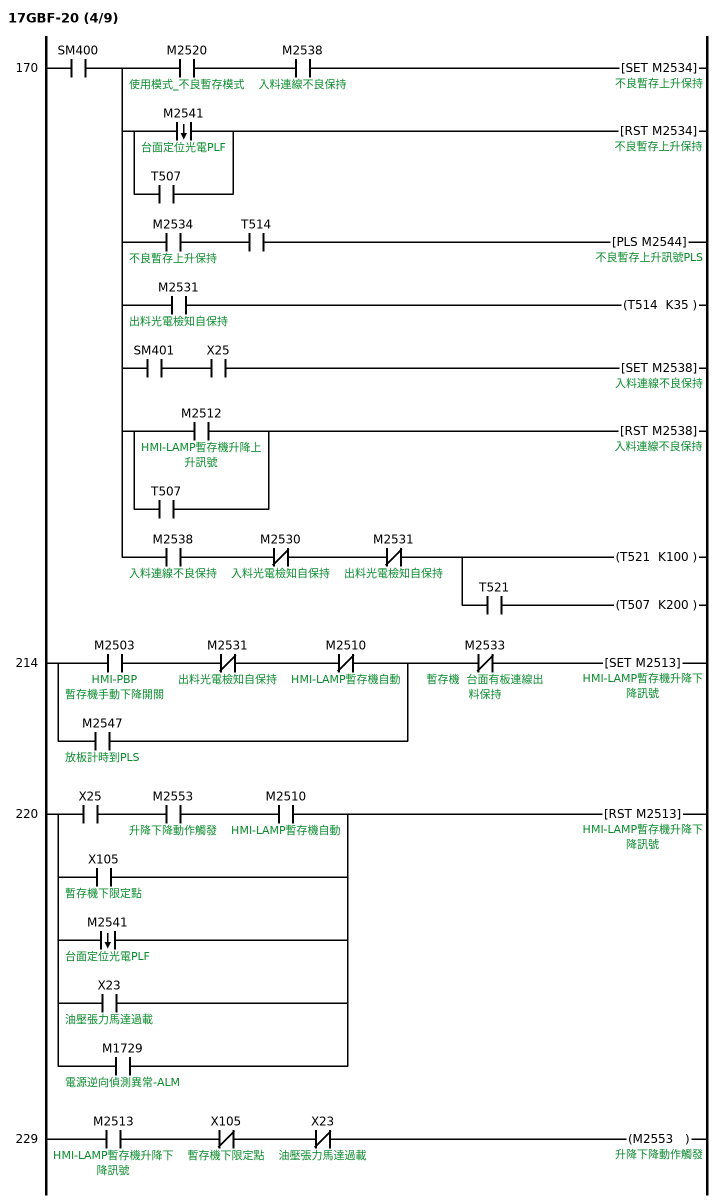
170   LD      SM400
      MPS
      AND     M2520  ; 使用模式_不良暫存模式
      AND     M2538  ; 入料連線不良保持
      SET     M2534  ; 不良暫存上升保持
      MRD
      LDF     M2541  ; 台面定位光電PLF
      OR      T507
      ANB
      RST     M2534  ; 不良暫存上升保持
      MRD
      AND     M2534  ; 不良暫存上升保持
      AND     T514
      PLS     M2544  ; 不良暫存上升訊號PLS
      MRD
      AND     M2531  ; 出料光電檢知自保持
      OUT     T514 K35
      MRD
      AND     SM401
      AND     X25
      SET     M2538  ; 入料連線不良保持
      MRD
      LD      M2512  ; HMI-LAMP暫存機升降上升訊號
      OR      T507
      ANB
      RST     M2538  ; 入料連線不良保持
      MPP
      AND     M2538  ; 入料連線不良保持
      ANI     M2530  ; 入料光電檢知自保持
      ANI     M2531  ; 出料光電檢知自保持
      OUT     T521 K100
      AND     T521
      OUT     T507 K200
214   LD      M2503  ; HMI-PBP 暫存機手動下降開關
      ANI     M2531  ; 出料光電檢知自保持
      ANI     M2510  ; HMI-LAMP暫存機自動
      OR      M2547  ; 放板計時到PLS
      ANI     M2533  ; 暫存機  台面有板連線出料保持
      SET     M2513  ; HMI-LAMP暫存機升降下降訊號
220   LD      X25
      AND     M2553  ; 升降下降動作觸發
      AND     M2510  ; HMI-LAMP暫存機自動
      OR      X105  ; 暫存機下限定點
      ORF     M2541  ; 台面定位光電PLF
      OR      X23  ; 油壓張力馬達過載
      OR      M1729  ; 電源逆向偵測異常-ALM
      RST     M2513  ; HMI-LAMP暫存機升降下降訊號
229   LD      M2513  ; HMI-LAMP暫存機升降下降訊號
      ANI     X105  ; 暫存機下限定點
      ANI     X23  ; 油壓張力馬達過載
      OUT     M2553  ; 升降下降動作觸發
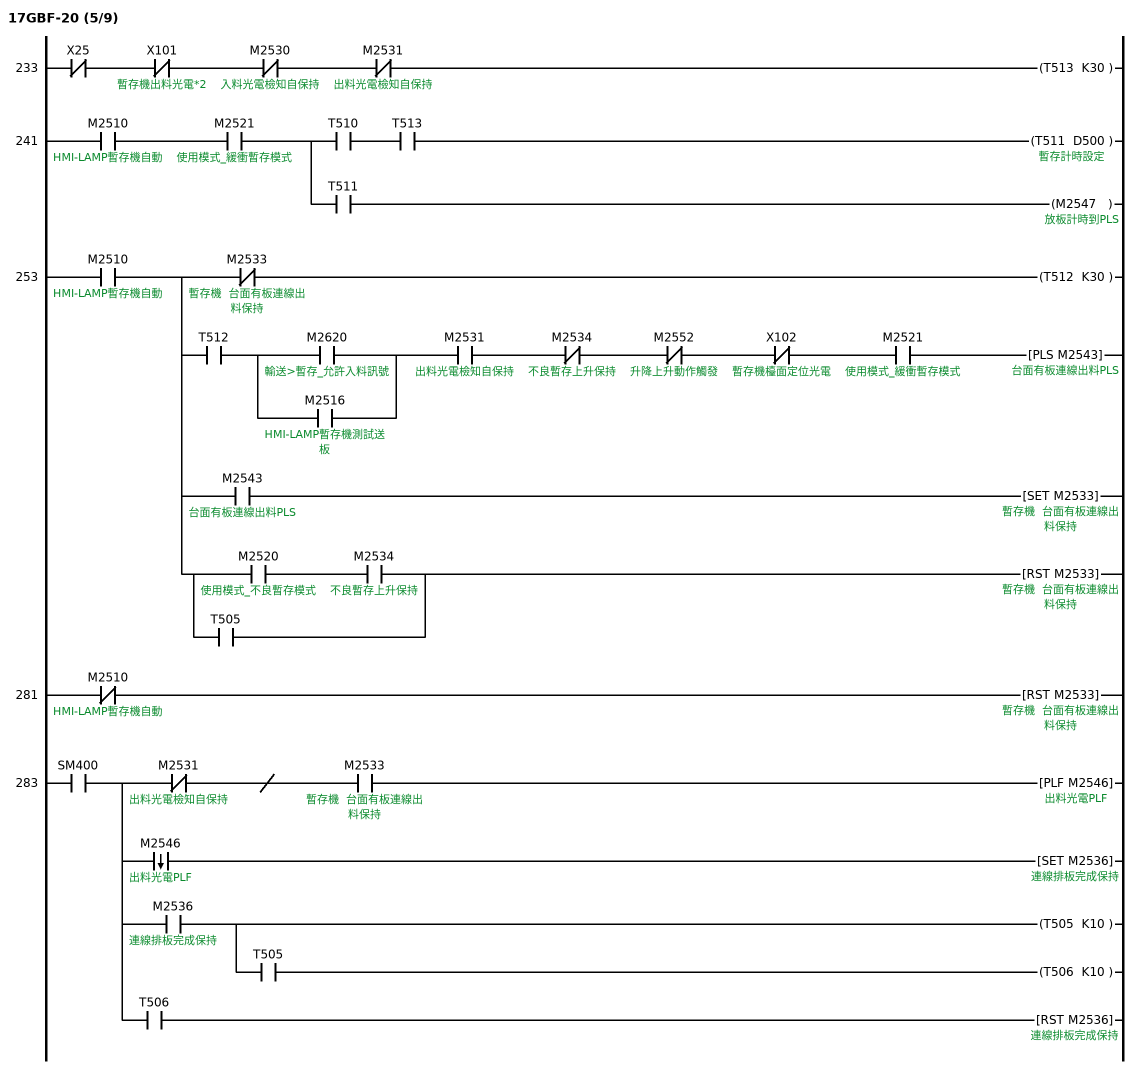
233   LDI     X25
      ANI     X101  ; 暫存機出料光電*2
      ANI     M2530  ; 入料光電檢知自保持
      ANI     M2531  ; 出料光電檢知自保持
      OUT     T513 K30
241   LD      M2510  ; HMI-LAMP暫存機自動
      AND     M2521  ; 使用模式_緩衝暫存模式
      MPS
      AND     T510
      AND     T513
      OUT     T511 D500  ; 暫存計時設定
      MPP
      AND     T511
      OUT     M2547  ; 放板計時到PLS
253   LD      M2510  ; HMI-LAMP暫存機自動
      MPS
      ANI     M2533  ; 暫存機  台面有板連線出料保持
      OUT     T512 K30
      MRD
      AND     T512
      LD      M2620  ; 輸送>暫存_允許入料訊號
      OR      M2516  ; HMI-LAMP暫存機測試送板
      ANB
      AND     M2531  ; 出料光電檢知自保持
      ANI     M2534  ; 不良暫存上升保持
      ANI     M2552  ; 升降上升動作觸發
      ANI     X102  ; 暫存機檯面定位光電
      AND     M2521  ; 使用模式_緩衝暫存模式
      PLS     M2543  ; 台面有板連線出料PLS
      MRD
      AND     M2543  ; 台面有板連線出料PLS
      SET     M2533  ; 暫存機  台面有板連線出料保持
      MPP
      LD      M2520  ; 使用模式_不良暫存模式
      AND     M2534  ; 不良暫存上升保持
      OR      T505
      ANB
      RST     M2533  ; 暫存機  台面有板連線出料保持
281   LDI     M2510  ; HMI-LAMP暫存機自動
      RST     M2533  ; 暫存機  台面有板連線出料保持
283   LD      SM400
      MPS
      ANI     M2531  ; 出料光電檢知自保持
      INV
      AND     M2533  ; 暫存機  台面有板連線出料保持
      PLF     M2546  ; 出料光電PLF
      MRD
      ANDF    M2546  ; 出料光電PLF
      SET     M2536  ; 連線排板完成保持
      MRD
      AND     M2536  ; 連線排板完成保持
      OUT     T505 K10
      AND     T505
      OUT     T506 K10
      MPP
      AND     T506
      RST     M2536  ; 連線排板完成保持
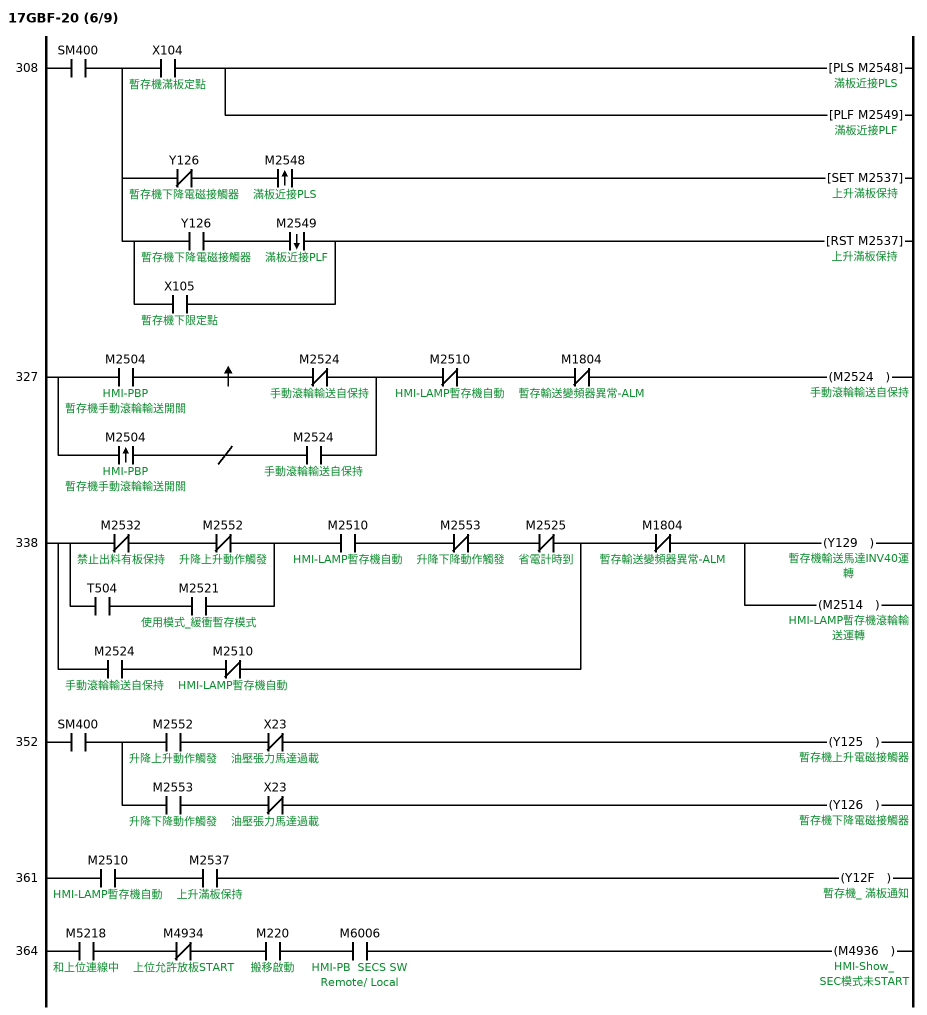
308   LD      SM400
      MPS
      AND     X104  ; 暫存機滿板定點
      PLS     M2548  ; 滿板近接PLS
      PLF     M2549  ; 滿板近接PLF
      MRD
      ANI     Y126  ; 暫存機下降電磁接觸器
      ANDP    M2548  ; 滿板近接PLS
      SET     M2537  ; 上升滿板保持
      MPP
      LD      Y126  ; 暫存機下降電磁接觸器
      ANDF    M2549  ; 滿板近接PLF
      OR      X105  ; 暫存機下限定點
      ANB
      RST     M2537  ; 上升滿板保持
327   LD      M2504  ; HMI-PBP 暫存機手動滾輪輸送開關
      MEP
      ANI     M2524  ; 手動滾輪輸送自保持
      LDP     M2504  ; HMI-PBP 暫存機手動滾輪輸送開關
      INV
      AND     M2524  ; 手動滾輪輸送自保持
      ORB
      ANI     M2510  ; HMI-LAMP暫存機自動
      ANI     M1804  ; 暫存輸送變頻器異常-ALM
      OUT     M2524  ; 手動滾輪輸送自保持
338   LDI     M2532  ; 禁止出料有板保持
      ANI     M2552  ; 升降上升動作觸發
      LD      T504
      AND     M2521  ; 使用模式_緩衝暫存模式
      ORB
      AND     M2510  ; HMI-LAMP暫存機自動
      ANI     M2553  ; 升降下降動作觸發
      ANI     M2525  ; 省電計時到
      LD      M2524  ; 手動滾輪輸送自保持
      ANI     M2510  ; HMI-LAMP暫存機自動
      ORB
      ANI     M1804  ; 暫存輸送變頻器異常-ALM
      OUT     Y129  ; 暫存機輸送馬達INV40運轉
      OUT     M2514  ; HMI-LAMP暫存機滾輪輸送運轉
352   LD      SM400
      MPS
      AND     M2552  ; 升降上升動作觸發
      ANI     X23  ; 油壓張力馬達過載
      OUT     Y125  ; 暫存機上升電磁接觸器
      MPP
      AND     M2553  ; 升降下降動作觸發
      ANI     X23  ; 油壓張力馬達過載
      OUT     Y126  ; 暫存機下降電磁接觸器
361   LD      M2510  ; HMI-LAMP暫存機自動
      AND     M2537  ; 上升滿板保持
      OUT     Y12F  ; 暫存機_ 滿板通知
364   LD      M5218  ; 和上位連線中
      ANI     M4934  ; 上位允許放板START
      AND     M220  ; 搬移啟動
      AND     M6006  ; HMI-PB  SECS SW  Remote/ Local
      OUT     M4936  ; HMI-Show_SEC模式未START
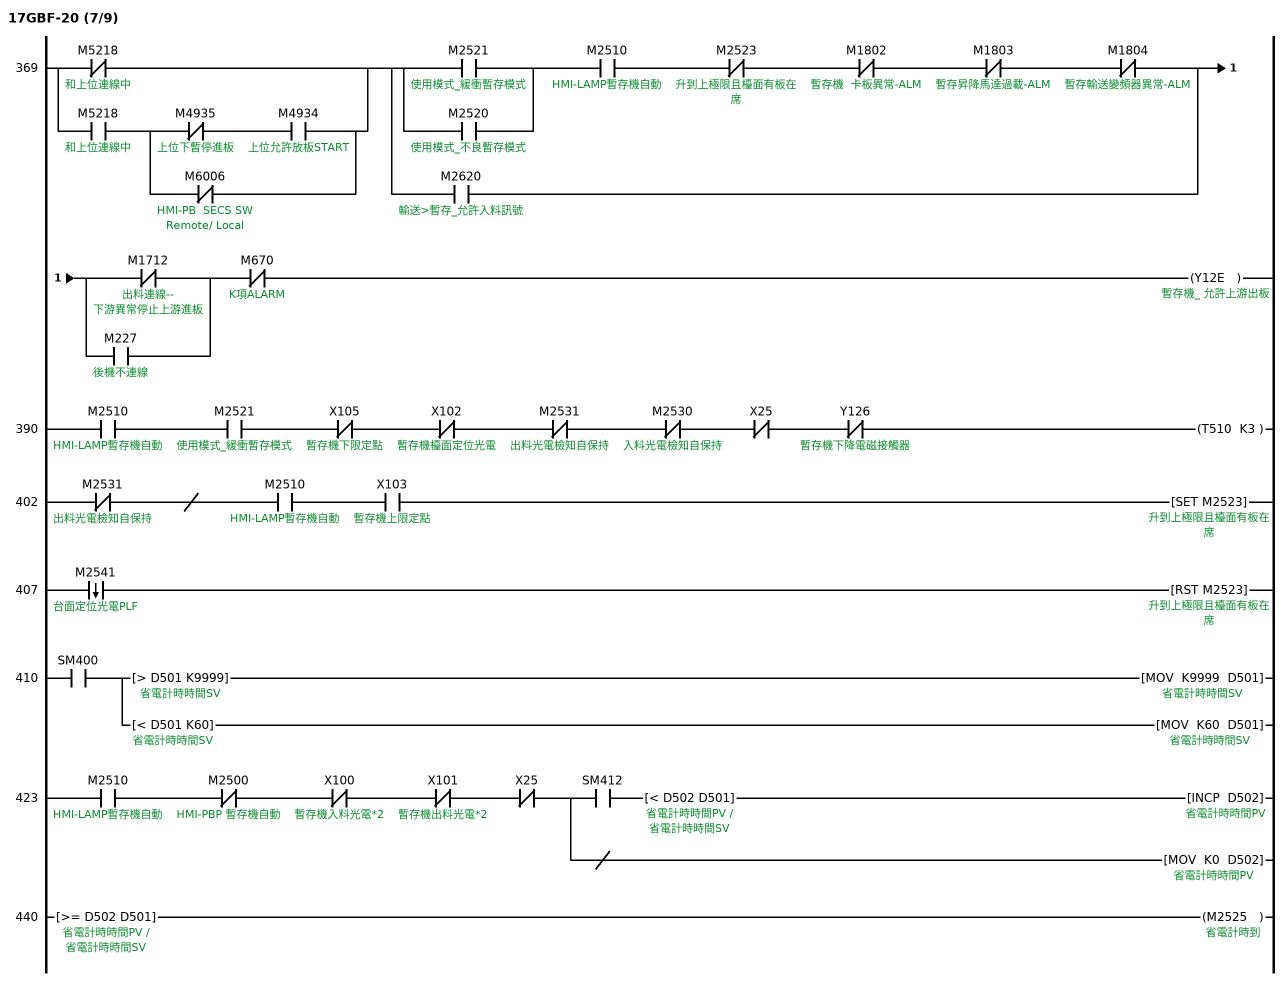
369   LDI     M5218  ; 和上位連線中
      LD      M5218  ; 和上位連線中
      LDI     M4935  ; 上位下暫停進板
      AND     M4934  ; 上位允許放板START
      ORI     M6006  ; HMI-PB  SECS SW  Remote/ Local
      ANB
      ORB
      LD      M2521  ; 使用模式_緩衝暫存模式
      OR      M2520  ; 使用模式_不良暫存模式
      AND     M2510  ; HMI-LAMP暫存機自動
      ANI     M2523  ; 升到上極限且檯面有板在席
      ANI     M1802  ; 暫存機  卡板異常-ALM
      ANI     M1803  ; 暫存昇降馬達過載-ALM
      ANI     M1804  ; 暫存輸送變頻器異常-ALM
      OR      M2620  ; 輸送>暫存_允許入料訊號
      ANB
      LDI     M1712  ; 出料連線--下游異常停止上游進板
      OR      M227  ; 後機不連線
      ANB
      ANI     M670  ; K項ALARM
      OUT     Y12E  ; 暫存機_ 允許上游出板
390   LD      M2510  ; HMI-LAMP暫存機自動
      AND     M2521  ; 使用模式_緩衝暫存模式
      ANI     X105  ; 暫存機下限定點
      ANI     X102  ; 暫存機檯面定位光電
      ANI     M2531  ; 出料光電檢知自保持
      ANI     M2530  ; 入料光電檢知自保持
      ANI     X25
      ANI     Y126  ; 暫存機下降電磁接觸器
      OUT     T510 K3
402   LDI     M2531  ; 出料光電檢知自保持
      INV
      AND     M2510  ; HMI-LAMP暫存機自動
      AND     X103  ; 暫存機上限定點
      SET     M2523  ; 升到上極限且檯面有板在席
407   LDF     M2541  ; 台面定位光電PLF
      RST     M2523  ; 升到上極限且檯面有板在席
410   LD      SM400
      MPS
      AND>    D501 K9999  ; 省電計時時間SV
      MOV     K9999 D501
      MPP
      AND<    D501 K60  ; 省電計時時間SV
      MOV     K60 D501
423   LD      M2510  ; HMI-LAMP暫存機自動
      ANI     M2500  ; HMI-PBP 暫存機自動
      ANI     X100  ; 暫存機入料光電*2
      ANI     X101  ; 暫存機出料光電*2
      ANI     X25
      MPS
      AND     SM412
      AND<    D502 D501  ; 省電計時時間PV / 省電計時時間SV
      INCP    D502
      MPP
      INV
      MOV     K0 D502
440   LD>=    D502 D501  ; 省電計時時間PV / 省電計時時間SV
      OUT     M2525  ; 省電計時到
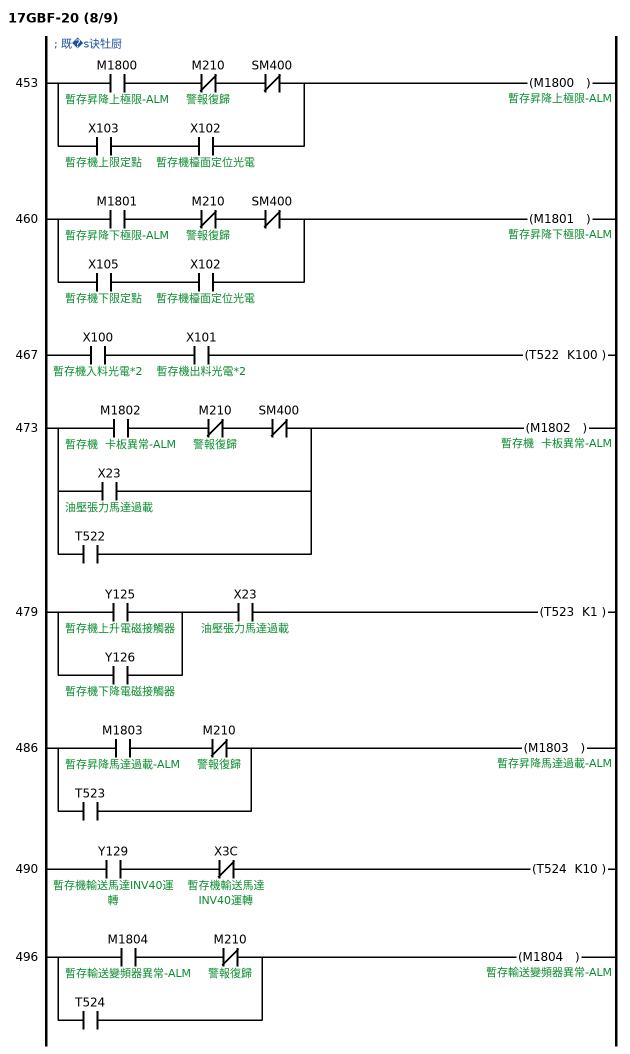
; 暫存機警報
453   LD      M1800  ; 暫存昇降上極限-ALM
      ANI     M210  ; 警報復歸
      ANI     SM400
      LD      X103  ; 暫存機上限定點
      AND     X102  ; 暫存機檯面定位光電
      ORB
      OUT     M1800  ; 暫存昇降上極限-ALM
460   LD      M1801  ; 暫存昇降下極限-ALM
      ANI     M210  ; 警報復歸
      ANI     SM400
      LD      X105  ; 暫存機下限定點
      AND     X102  ; 暫存機檯面定位光電
      ORB
      OUT     M1801  ; 暫存昇降下極限-ALM
467   LD      X100  ; 暫存機入料光電*2
      AND     X101  ; 暫存機出料光電*2
      OUT     T522 K100
473   LD      M1802  ; 暫存機  卡板異常-ALM
      ANI     M210  ; 警報復歸
      ANI     SM400
      OR      X23  ; 油壓張力馬達過載
      OR      T522
      OUT     M1802  ; 暫存機  卡板異常-ALM
479   LD      Y125  ; 暫存機上升電磁接觸器
      OR      Y126  ; 暫存機下降電磁接觸器
      AND     X23  ; 油壓張力馬達過載
      OUT     T523 K1
486   LD      M1803  ; 暫存昇降馬達過載-ALM
      ANI     M210  ; 警報復歸
      OR      T523
      OUT     M1803  ; 暫存昇降馬達過載-ALM
490   LD      Y129  ; 暫存機輸送馬達INV40運轉
      ANI     X3C  ; 暫存機輸送馬達  INV40運轉
      OUT     T524 K10
496   LD      M1804  ; 暫存輸送變頻器異常-ALM
      ANI     M210  ; 警報復歸
      OR      T524
      OUT     M1804  ; 暫存輸送變頻器異常-ALM
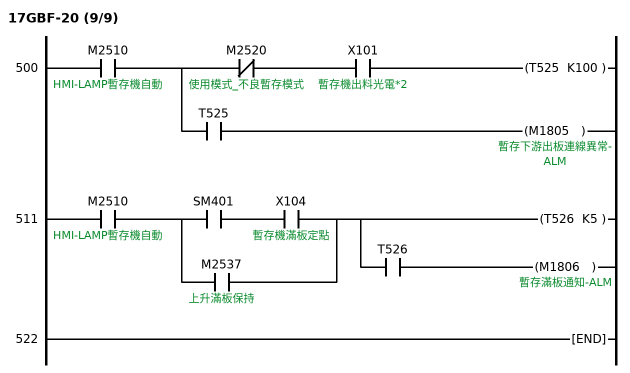
500   LD      M2510  ; HMI-LAMP暫存機自動
      MPS
      ANI     M2520  ; 使用模式_不良暫存模式
      AND     X101  ; 暫存機出料光電*2
      OUT     T525 K100
      MPP
      AND     T525
      OUT     M1805  ; 暫存下游出板連線異常-ALM
511   LD      M2510  ; HMI-LAMP暫存機自動
      LD      SM401
      AND     X104  ; 暫存機滿板定點
      OR      M2537  ; 上升滿板保持
      ANB
      OUT     T526 K5
      AND     T526
      OUT     M1806  ; 暫存滿板通知-ALM
522   END
END_PROGRAM

PROGRAM 18GCV
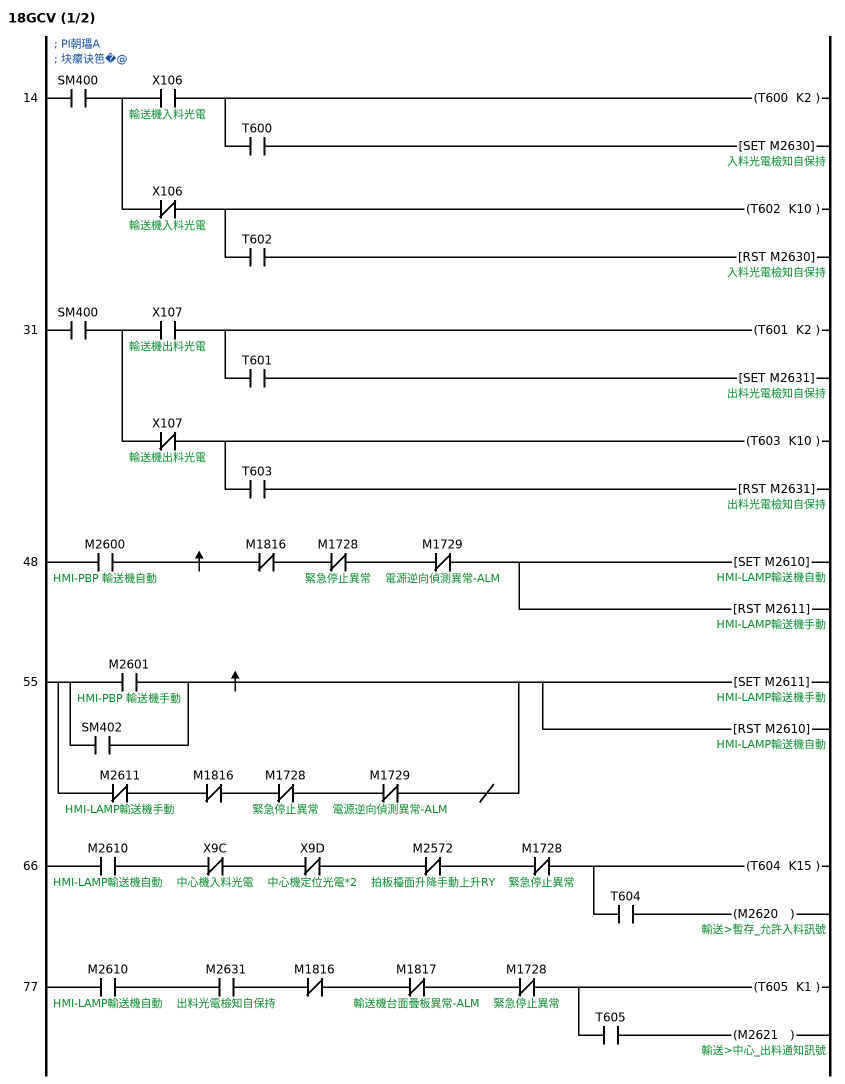
; PI朝瓃Α
; 輸送機動作
14    LD      SM400
      MPS
      AND     X106  ; 輸送機入料光電
      OUT     T600 K2
      AND     T600
      SET     M2630  ; 入料光電檢知自保持
      MPP
      ANI     X106  ; 輸送機入料光電
      OUT     T602 K10
      AND     T602
      RST     M2630  ; 入料光電檢知自保持
31    LD      SM400
      MPS
      AND     X107  ; 輸送機出料光電
      OUT     T601 K2
      AND     T601
      SET     M2631  ; 出料光電檢知自保持
      MPP
      ANI     X107  ; 輸送機出料光電
      OUT     T603 K10
      AND     T603
      RST     M2631  ; 出料光電檢知自保持
48    LD      M2600  ; HMI-PBP 輸送機自動
      MEP
      ANI     M1816
      ANI     M1728  ; 緊急停止異常
      ANI     M1729  ; 電源逆向偵測異常-ALM
      SET     M2610  ; HMI-LAMP輸送機自動
      RST     M2611  ; HMI-LAMP輸送機手動
55    LD      M2601  ; HMI-PBP 輸送機手動
      OR      SM402
      MEP
      LDI     M2611  ; HMI-LAMP輸送機手動
      ANI     M1816
      ANI     M1728  ; 緊急停止異常
      ANI     M1729  ; 電源逆向偵測異常-ALM
      INV
      ORB
      SET     M2611  ; HMI-LAMP輸送機手動
      RST     M2610  ; HMI-LAMP輸送機自動
66    LD      M2610  ; HMI-LAMP輸送機自動
      ANI     X9C  ; 中心機入料光電
      ANI     X9D  ; 中心機定位光電*2
      ANI     M2572  ; 拍板檯面升降手動上升RY
      ANI     M1728  ; 緊急停止異常
      OUT     T604 K15
      AND     T604
      OUT     M2620  ; 輸送>暫存_允許入料訊號
77    LD      M2610  ; HMI-LAMP輸送機自動
      AND     M2631  ; 出料光電檢知自保持
      ANI     M1816
      ANI     M1817  ; 輸送機台面疊板異常-ALM
      ANI     M1728  ; 緊急停止異常
      OUT     T605 K1
      AND     T605
      OUT     M2621  ; 輸送>中心_出料通知訊號
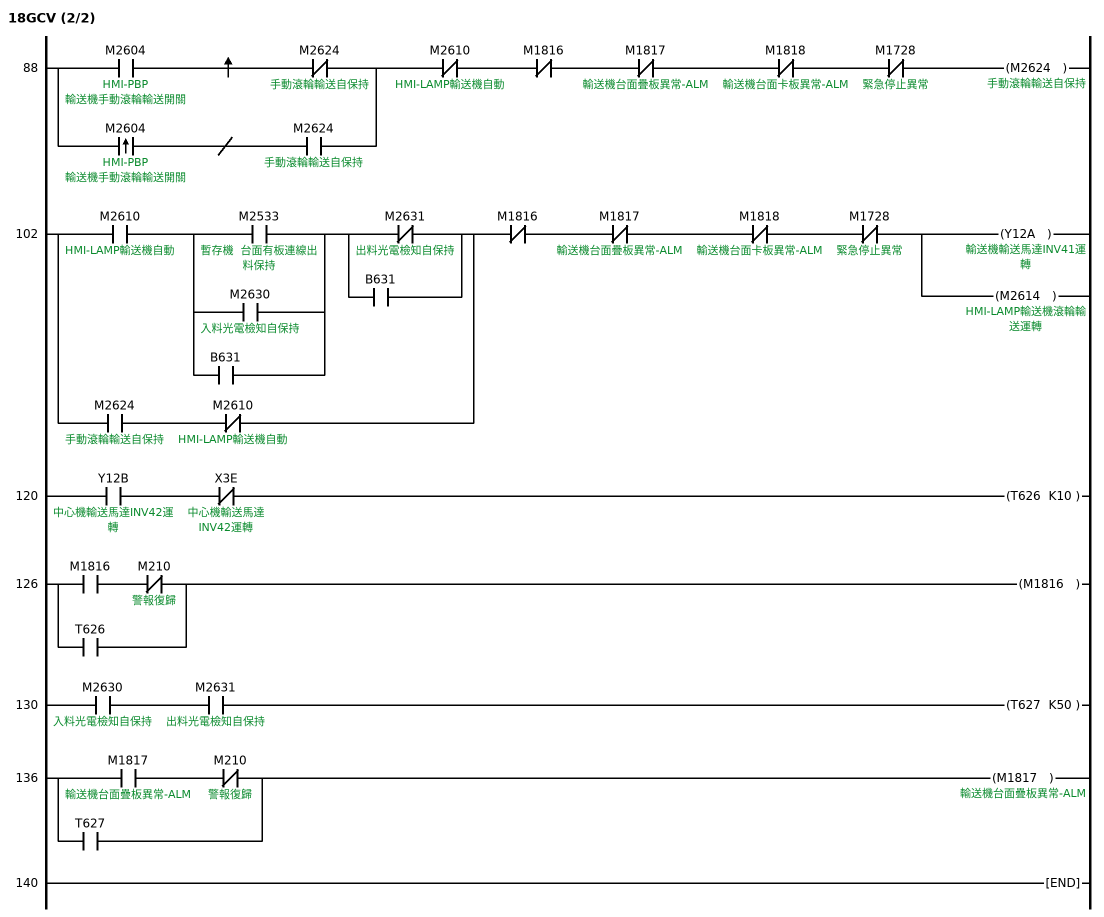
88    LD      M2604  ; HMI-PBP 輸送機手動滾輪輸送開關
      MEP
      ANI     M2624  ; 手動滾輪輸送自保持
      LDP     M2604  ; HMI-PBP 輸送機手動滾輪輸送開關
      INV
      AND     M2624  ; 手動滾輪輸送自保持
      ORB
      ANI     M2610  ; HMI-LAMP輸送機自動
      ANI     M1816
      ANI     M1817  ; 輸送機台面疊板異常-ALM
      ANI     M1818  ; 輸送機台面卡板異常-ALM
      ANI     M1728  ; 緊急停止異常
      OUT     M2624  ; 手動滾輪輸送自保持
102   LD      M2610  ; HMI-LAMP輸送機自動
      LD      M2533  ; 暫存機  台面有板連線出料保持
      OR      M2630  ; 入料光電檢知自保持
      OR      B631
      ANB
      LDI     M2631  ; 出料光電檢知自保持
      OR      B631
      ANB
      LD      M2624  ; 手動滾輪輸送自保持
      ANI     M2610  ; HMI-LAMP輸送機自動
      ORB
      ANI     M1816
      ANI     M1817  ; 輸送機台面疊板異常-ALM
      ANI     M1818  ; 輸送機台面卡板異常-ALM
      ANI     M1728  ; 緊急停止異常
      OUT     Y12A  ; 輸送機輸送馬達INV41運轉
      OUT     M2614  ; HMI-LAMP輸送機滾輪輸送運轉
120   LD      Y12B  ; 中心機輸送馬達INV42運轉
      ANI     X3E  ; 中心機輸送馬達  INV42運轉
      OUT     T626 K10
126   LD      M1816
      ANI     M210  ; 警報復歸
      OR      T626
      OUT     M1816
130   LD      M2630  ; 入料光電檢知自保持
      AND     M2631  ; 出料光電檢知自保持
      OUT     T627 K50
136   LD      M1817  ; 輸送機台面疊板異常-ALM
      ANI     M210  ; 警報復歸
      OR      T627
      OUT     M1817  ; 輸送機台面疊板異常-ALM
140   END
END_PROGRAM

PROGRAM 19GTC-7
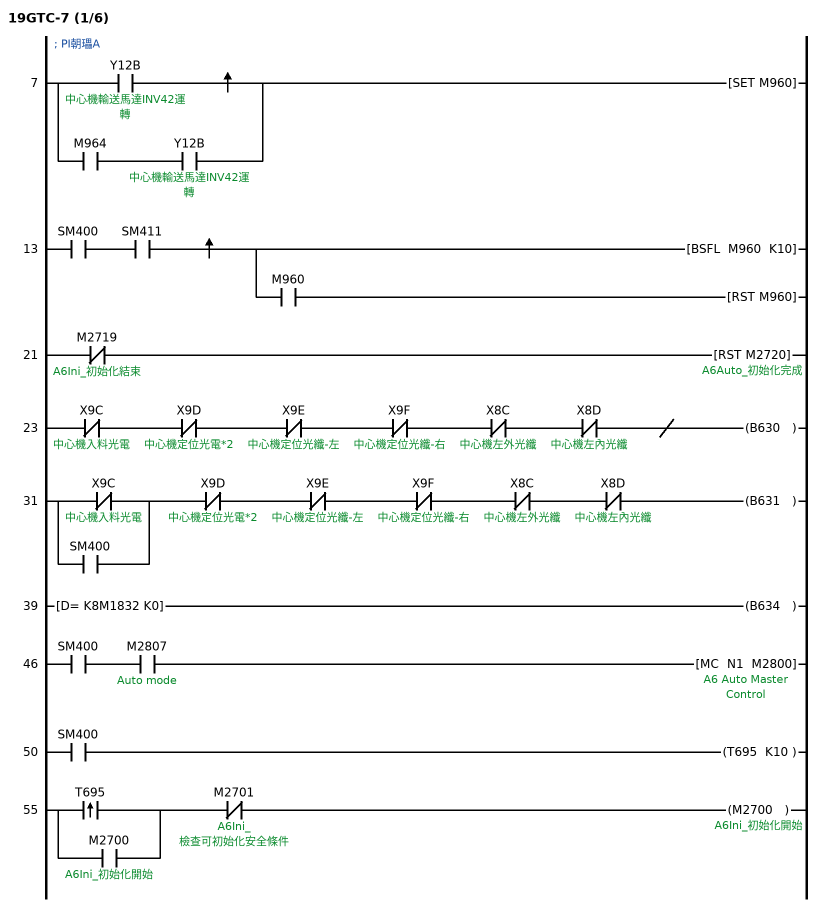
; PI朝瓃Α
7     LD      Y12B  ; 中心機輸送馬達INV42運轉
      MEP
      LD      M964
      AND     Y12B  ; 中心機輸送馬達INV42運轉
      ORB
      SET     M960
13    LD      SM400
      AND     SM411
      MEP
      BSFL    M960 K10
      AND     M960
      RST     M960
21    LDI     M2719  ; A6Ini_初始化結束
      RST     M2720  ; A6Auto_初始化完成
23    LDI     X9C  ; 中心機入料光電
      ANI     X9D  ; 中心機定位光電*2
      ANI     X9E  ; 中心機定位光纖-左
      ANI     X9F  ; 中心機定位光纖-右
      ANI     X8C  ; 中心機左外光纖
      ANI     X8D  ; 中心機左內光纖
      INV
      OUT     B630
31    LDI     X9C  ; 中心機入料光電
      OR      SM400
      ANI     X9D  ; 中心機定位光電*2
      ANI     X9E  ; 中心機定位光纖-左
      ANI     X9F  ; 中心機定位光纖-右
      ANI     X8C  ; 中心機左外光纖
      ANI     X8D  ; 中心機左內光纖
      OUT     B631
39    LDD=    K8M1832 K0
      OUT     B634
46    LD      SM400
      AND     M2807  ; Auto mode
      MC      N1 M2800  ; A6 Auto Master Control
50    LD      SM400
      OUT     T695 K10
55    LDP     T695
      OR      M2700  ; A6Ini_初始化開始
      ANI     M2701  ; A6Ini_檢查可初始化安全條件
      OUT     M2700  ; A6Ini_初始化開始
